QRS_NEXT_CUT()
PTP {E1 29336.867,E2 29336.867}
PTP {X 0,Y 607.919,A -85,B 0,C 180,E1 29336.867,E2 29336.867,E3 0,E4 0,E5 0,E6 0}
QRS_SPEED_INIT()
LIN {X 0,Y 607.919,Z 1319.5,A -85,B 0,C 180,E1 29336.867,E2 29336.867,E3 0,E4 0,E5 0,E6 0} C_VEL
LIN {X 0,Y 607.919,Z 669.088,A -85,B 0,C 180,E1 29336.867,E2 29336.867} C_VEL
LIN {X 0,Y 607.919,Z 661.015,A -85,B 0,C 180,E1 29336.867,E2 29336.867} C_VEL
LIN {X 0,Y 607.916,Z 659.015,A -85,B 0,C 180,E1 29336.679,E2 29336.679} C_VEL
LIN {X 0,Y 607.893,Z 659.005,A -85,B 0,C 180,E1 29333.483,E2 29333.483} C_VEL
LIN {X 0,Y 607.909,Z 659.016,A -85,B 0,C 180,E1 29330.342,E2 29330.342} C_VEL
LIN {X 0,Y 607.894,Z 659.005,A -85,B 0,C 180,E1 29327.171,E2 29327.171} C_VEL
LIN {X 0,Y 607.91,Z 659.015,A -85,B 0,C 180,E1 29323.959,E2 29323.959} C_VEL
LIN {X 0,Y 607.895,Z 659.005,A -85,B 0,C 180,E1 29320.748,E2 29320.748} C_VEL
LIN {X 0,Y 607.917,Z 659.014,A -85,B 0,C 180,E1 29317.564,E2 29317.564} C_VEL
LIN {X 0,Y 607.897,Z 659.005,A -85,B 0,C 180,E1 29314.331,E2 29314.331} C_VEL
LIN {X 0,Y 607.917,Z 659.013,A -85,B 0,C 180,E1 29311.19,E2 29311.19} C_VEL
LIN {X 0,Y 607.905,Z 659.003,A -85,B 0,C 180,E1 29308.021,E2 29308.021} C_VEL
LIN {X 0,Y 607.915,Z 659.014,A -85,B 0,C 180,E1 29304.826,E2 29304.826} C_VEL
LIN {X 0,Y 607.905,Z 659.004,A -85,B 0,C 180,E1 29301.558,E2 29301.558} C_VEL
LIN {X 0,Y 607.904,Z 659.011,A -85,B 0,C 180,E1 29298.305,E2 29298.305} C_VEL
LIN {X 0,Y 607.908,Z 659.004,A -85,B 0,C 180,E1 29295.122,E2 29295.122} C_VEL
LIN {X 0,Y 607.908,Z 659.011,A -85,B 0,C 180,E1 29291.894,E2 29291.894} C_VEL
LIN {X 0,Y 607.911,Z 659.003,A -85,B 0,C 180,E1 29288.681,E2 29288.681} C_VEL
LIN {X 0,Y 607.908,Z 659.008,A -85,B 0,C 180,E1 29285.491,E2 29285.491} C_VEL
LIN {X 0,Y 607.91,Z 658.993,A -85,B 0,C 180,E1 29282.285,E2 29282.285} C_VEL
LIN {X 0,Y 607.909,Z 659.344,A -85,B 0,C 180,E1 29281.725,E2 29281.725} C_VEL
LIN {X 0,Y 607.912,Z 660.667,A -85,B 0,C 180,E1 29281.627,E2 29281.627} C_VEL
LIN {X 0,Y 607.912,Z 878.758,A -85,B 0,C 180,E1 29278.702,E2 29278.702} C_VEL
LIN {X 0,Y 607.912,Z 916.881,A -85,B 0,C 180,E1 29278.166,E2 29278.166} C_VEL
LIN {X 0,Y 607.906,Z 937.091,A -85,B 0,C 180,E1 29277.713,E2 29277.713} C_VEL
LIN {X 0,Y 607.913,Z 958.264,A -85,B 0,C 180,E1 29277.076,E2 29277.076} C_VEL
LIN {X 0,Y 607.913,Z 976.775,A -85,B 0,C 180,E1 29276.364,E2 29276.364} C_VEL
LIN {X 0,Y 607.919,Z 997.894,A -85,B 0,C 180,E1 29275.368,E2 29275.368} C_VEL
LIN {X 0,Y 607.917,Z 1017.228,A -85,B 0,C 180,E1 29274.278,E2 29274.278} C_VEL
LIN {X 0,Y 607.914,Z 1035.659,A -85,B 0,C 180,E1 29273.044,E2 29273.044} C_VEL
LIN {X 0,Y 607.916,Z 1053.23,A -85,B 0,C 180,E1 29271.678,E2 29271.678} C_VEL
LIN {X 0,Y 607.912,Z 1070.203,A -85,B 0,C 180,E1 29270.155,E2 29270.155} C_VEL
LIN {X 0,Y 607.917,Z 1086.083,A -85,B 0,C 180,E1 29268.507,E2 29268.507} C_VEL
LIN {X 0,Y 607.913,Z 1100.76,A -85,B 0,C 180,E1 29266.728,E2 29266.728} C_VEL
LIN {X 0,Y 607.912,Z 1113.249,A -85,B 0,C 180,E1 29264.964,E2 29264.964} C_VEL
LIN {X 0,Y 607.916,Z 1124.49,A -85,B 0,C 180,E1 29263.119,E2 29263.119} C_VEL
LIN {X 0,Y 607.902,Z 1133.845,A -85,B 0,C 180,E1 29261.287,E2 29261.287} C_VEL
LIN {X 0,Y 607.899,Z 1142.297,A -85,B 0,C 180,E1 29259.276,E2 29259.276} C_VEL
LIN {X 0,Y 607.904,Z 1148.818,A -85,B 0,C 180,E1 29257.345,E2 29257.345} C_VEL
LIN {X 0,Y 607.911,Z 1153.711,A -85,B 0,C 180,E1 29255.379,E2 29255.379} C_VEL
LIN {X 0,Y 607.918,Z 1157.29,A -85,B 0,C 180,E1 29253.292,E2 29253.292} C_VEL
LIN {X 0,Y 607.907,Z 1159.182,A -85,B 0,C 180,E1 29251.225,E2 29251.225} C_VEL
LIN {X 0,Y 607.898,Z 1159.339,A -85,B 0,C 180,E1 29249.246,E2 29249.246} C_VEL
LIN {X 0,Y 607.899,Z 1157.836,A -85,B 0,C 180,E1 29247.077,E2 29247.077} C_VEL
LIN {X 0,Y 607.896,Z 1154.903,A -85,B 0,C 180,E1 29245.094,E2 29245.094} C_VEL
LIN {X 0,Y 607.909,Z 1150.265,A -85,B 0,C 180,E1 29243.104,E2 29243.104} C_VEL
LIN {X 0,Y 607.917,Z 1144.051,A -85,B 0,C 180,E1 29241.106,E2 29241.106} C_VEL
LIN {X 0,Y 607.916,Z 1136.441,A -85,B 0,C 180,E1 29239.193,E2 29239.193} C_VEL
LIN {X 0,Y 607.909,Z 1126.947,A -85,B 0,C 180,E1 29237.249,E2 29237.249} C_VEL
LIN {X 0,Y 607.901,Z 1116.406,A -85,B 0,C 180,E1 29235.425,E2 29235.425} C_VEL
LIN {X 0,Y 607.906,Z 1104.361,A -85,B 0,C 180,E1 29233.665,E2 29233.665} C_VEL
LIN {X 0,Y 607.907,Z 1090.255,A -85,B 0,C 180,E1 29231.89,E2 29231.89} C_VEL
LIN {X 0,Y 607.908,Z 1075.163,A -85,B 0,C 180,E1 29230.246,E2 29230.246} C_VEL
LIN {X 0,Y 607.91,Z 1058.641,A -85,B 0,C 180,E1 29228.686,E2 29228.686} C_VEL
LIN {X 0,Y 607.915,Z 1041.052,A -85,B 0,C 180,E1 29227.263,E2 29227.263} C_VEL
LIN {X 0,Y 607.915,Z 1022.644,A -85,B 0,C 180,E1 29225.98,E2 29225.98} C_VEL
LIN {X 0,Y 607.918,Z 1003.587,A -85,B 0,C 180,E1 29224.84,E2 29224.84} C_VEL
LIN {X 0,Y 607.911,Z 984.81,A -85,B 0,C 180,E1 29223.901,E2 29223.901} C_VEL
LIN {X 0,Y 607.918,Z 963.681,A -85,B 0,C 180,E1 29223.03,E2 29223.03} C_VEL
LIN {X 0,Y 607.909,Z 943.544,A -85,B 0,C 180,E1 29222.367,E2 29222.367} C_VEL
LIN {X 0,Y 607.919,Z 923.855,A -85,B 0,C 180,E1 29221.888,E2 29221.888} C_VEL
LIN {X 0,Y 607.905,Z 902.891,A -85,B 0,C 180,E1 29221.526,E2 29221.526} C_VEL
LIN {X 0,Y 607.914,Z 678.859,A -85,B 0,C 180,E1 29218.535,E2 29218.535} C_VEL
LIN {X 0,Y 607.914,Z 659.964,A -85,B 0,C 180,E1 29218.261,E2 29218.261} C_VEL
LIN {X 0,Y 607.909,Z 659.135,A -85,B 0,C 180,E1 29218.133,E2 29218.133} C_VEL
LIN {X 0,Y 607.894,Z 659.003,A -85,B 0,C 180,E1 29215.084,E2 29215.084} C_VEL
LIN {X 0,Y 607.912,Z 659.013,A -85,B 0,C 180,E1 29211.92,E2 29211.92} C_VEL
LIN {X 0,Y 607.898,Z 659.005,A -85,B 0,C 180,E1 29208.735,E2 29208.735} C_VEL
LIN {X 0,Y 607.91,Z 659.013,A -85,B 0,C 180,E1 29205.522,E2 29205.522} C_VEL
LIN {X 0,Y 607.905,Z 659.002,A -85,B 0,C 180,E1 29202.398,E2 29202.398} C_VEL
LIN {X 0,Y 607.909,Z 659.013,A -85,B 0,C 180,E1 29199.167,E2 29199.167} C_VEL
LIN {X 0,Y 607.907,Z 659.003,A -85,B 0,C 180,E1 29195.957,E2 29195.957} C_VEL
LIN {X 0,Y 607.91,Z 659.012,A -85,B 0,C 180,E1 29192.76,E2 29192.76} C_VEL
LIN {X 0,Y 607.912,Z 659.002,A -85,B 0,C 180,E1 29189.537,E2 29189.537} C_VEL
LIN {X 0,Y 607.907,Z 659.01,A -85,B 0,C 180,E1 29186.26,E2 29186.26} C_VEL
LIN {X 0,Y 607.912,Z 659.004,A -85,B 0,C 180,E1 29183.045,E2 29183.045} C_VEL
LIN {X 0,Y 607.908,Z 659.008,A -85,B 0,C 180,E1 29179.805,E2 29179.805} C_VEL
LIN {X 0,Y 607.912,Z 659.005,A -85,B 0,C 180,E1 29176.63,E2 29176.63} C_VEL
LIN {X 0,Y 607.906,Z 659.007,A -85,B 0,C 180,E1 29173.313,E2 29173.313} C_VEL
LIN {X 0,Y 607.912,Z 659.008,A -85,B 0,C 180,E1 29170.041,E2 29170.041} C_VEL
LIN {X 0,Y 607.903,Z 659.005,A -85,B 0,C 180,E1 29166.801,E2 29166.801} C_VEL
LIN {X 0,Y 607.912,Z 659.009,A -85,B 0,C 180,E1 29163.583,E2 29163.583} C_VEL
LIN {X 0,Y 607.906,Z 659.005,A -85,B 0,C 180,E1 29160.377,E2 29160.377} C_VEL
LIN {X 0,Y 607.917,Z 659.011,A -85,B 0,C 180,E1 29157.078,E2 29157.078} C_VEL
LIN {X 0,Y 607.903,Z 659.004,A -85,B 0,C 180,E1 29153.863,E2 29153.863} C_VEL
LIN {X 0,Y 607.919,Z 659.013,A -85,B 0,C 180,E1 29150.629,E2 29150.629} C_VEL
LIN {X 0,Y 607.901,Z 659.003,A -85,B 0,C 180,E1 29147.364,E2 29147.364} C_VEL
LIN {X 0,Y 607.907,Z 659.015,A -85,B 0,C 180,E1 29144.156,E2 29144.156} C_VEL
LIN {X 0,Y 607.901,Z 659.004,A -85,B 0,C 180,E1 29140.895,E2 29140.895} C_VEL
LIN {X 0,Y 607.9,Z 659.013,A -85,B 0,C 180,E1 29137.67,E2 29137.67} C_VEL
LIN {X 0,Y 607.904,Z 659.004,A -85,B 0,C 180,E1 29134.474,E2 29134.474} C_VEL
LIN {X 0,Y 607.904,Z 659.011,A -85,B 0,C 180,E1 29131.239,E2 29131.239} C_VEL
LIN {X 0,Y 607.905,Z 659.005,A -85,B 0,C 180,E1 29128.021,E2 29128.021} C_VEL
LIN {X 0,Y 607.905,Z 659.011,A -85,B 0,C 180,E1 29124.827,E2 29124.827} C_VEL
LIN {X 0,Y 607.908,Z 659.004,A -85,B 0,C 180,E1 29121.677,E2 29121.677} C_VEL
LIN {X 0,Y 607.907,Z 659.006,A -85,B 0,C 180,E1 29118.358,E2 29118.358} C_VEL
LIN {X 0,Y 607.909,Z 659.006,A -85,B 0,C 180,E1 29115.143,E2 29115.143} C_VEL
LIN {X 0,Y 607.908,Z 659.008,A -85,B 0,C 180,E1 29111.894,E2 29111.894} C_VEL
LIN {X 0,Y 607.909,Z 659.002,A -85,B 0,C 180,E1 29108.681,E2 29108.681} C_VEL
LIN {X 0,Y 607.899,Z 659.315,A -85,B 0,C 180,E1 29108.411,E2 29108.411} C_VEL
LIN {X 0,Y 607.916,Z 664.975,A -85,B 0,C 180,E1 29108.018,E2 29108.018} C_VEL
LIN {X 0,Y 607.893,Z 712.988,A -85,B 0,C 180,E1 29105.088,E2 29105.088} C_VEL
LIN {X 0,Y 607.911,Z 759.172,A -85,B 0,C 180,E1 29102.374,E2 29102.374} C_VEL
LIN {X 0,Y 607.916,Z 982.293,A -85,B 0,C 180,E1 29099.362,E2 29099.362} C_VEL
LIN {X 0,Y 607.907,Z 1064.715,A -85,B 0,C 180,E1 29098.246,E2 29098.246} C_VEL
LIN {X 0,Y 607.91,Z 1085.231,A -85,B 0,C 180,E1 29097.805,E2 29097.805} C_VEL
LIN {X 0,Y 607.91,Z 1105.827,A -85,B 0,C 180,E1 29097.208,E2 29097.208} C_VEL
LIN {X 0,Y 607.905,Z 1126.592,A -85,B 0,C 180,E1 29096.417,E2 29096.417} C_VEL
LIN {X 0,Y 607.918,Z 1147.757,A -85,B 0,C 180,E1 29095.421,E2 29095.421} C_VEL
LIN {X 0,Y 607.916,Z 1167.098,A -85,B 0,C 180,E1 29094.332,E2 29094.332} C_VEL
LIN {X 0,Y 607.914,Z 1185.57,A -85,B 0,C 180,E1 29093.095,E2 29093.095} C_VEL
LIN {X 0,Y 607.913,Z 1203.763,A -85,B 0,C 180,E1 29091.678,E2 29091.678} C_VEL
LIN {X 0,Y 607.915,Z 1220.656,A -85,B 0,C 180,E1 29090.155,E2 29090.155} C_VEL
LIN {X 0,Y 607.918,Z 1236.469,A -85,B 0,C 180,E1 29088.507,E2 29088.507} C_VEL
LIN {X 0,Y 607.913,Z 1250.41,A -85,B 0,C 180,E1 29086.817,E2 29086.817} C_VEL
LIN {X 0,Y 607.918,Z 1262.904,A -85,B 0,C 180,E1 29085.062,E2 29085.062} C_VEL
LIN {X 0,Y 607.918,Z 1274.422,A -85,B 0,C 180,E1 29083.176,E2 29083.176} C_VEL
LIN {X 0,Y 607.908,Z 1284.062,A -85,B 0,C 180,E1 29081.287,E2 29081.287} C_VEL
LIN {X 0,Y 607.907,Z 1292.364,A -85,B 0,C 180,E1 29079.302,E2 29079.302} C_VEL
LIN {X 0,Y 607.909,Z 1298.926,A -85,B 0,C 180,E1 29077.351,E2 29077.351} C_VEL
LIN {X 0,Y 607.915,Z 1303.809,A -85,B 0,C 180,E1 29075.379,E2 29075.379} C_VEL
LIN {X 0,Y 607.916,Z 1307.446,A -85,B 0,C 180,E1 29073.206,E2 29073.206} C_VEL
LIN {X 0,Y 607.91,Z 1309.21,A -85,B 0,C 180,E1 29071.225,E2 29071.225} C_VEL
LIN {X 0,Y 607.897,Z 1309.329,A -85,B 0,C 180,E1 29069.246,E2 29069.246} C_VEL
LIN {X 0,Y 607.897,Z 1307.895,A -85,B 0,C 180,E1 29067.172,E2 29067.172} C_VEL
LIN {X 0,Y 607.902,Z 1304.987,A -85,B 0,C 180,E1 29065.188,E2 29065.188} C_VEL
LIN {X 0,Y 607.912,Z 1300.398,A -85,B 0,C 180,E1 29063.199,E2 29063.199} C_VEL
LIN {X 0,Y 607.909,Z 1294.238,A -85,B 0,C 180,E1 29061.202,E2 29061.202} C_VEL
LIN {X 0,Y 607.909,Z 1286.657,A -85,B 0,C 180,E1 29059.289,E2 29059.289} C_VEL
LIN {X 0,Y 607.9,Z 1277.328,A -85,B 0,C 180,E1 29057.364,E2 29057.364} C_VEL
LIN {X 0,Y 607.901,Z 1266.747,A -85,B 0,C 180,E1 29055.523,E2 29055.523} C_VEL
LIN {X 0,Y 607.913,Z 1254.744,A -85,B 0,C 180,E1 29053.764,E2 29053.764} C_VEL
LIN {X 0,Y 607.911,Z 1240.72,A -85,B 0,C 180,E1 29051.989,E2 29051.989} C_VEL
LIN {X 0,Y 607.908,Z 1225.72,A -85,B 0,C 180,E1 29050.346,E2 29050.346} C_VEL
LIN {X 0,Y 607.912,Z 1208.705,A -85,B 0,C 180,E1 29048.737,E2 29048.737} C_VEL
LIN {X 0,Y 607.919,Z 1191.227,A -85,B 0,C 180,E1 29047.322,E2 29047.322} C_VEL
LIN {X 0,Y 607.915,Z 1172.745,A -85,B 0,C 180,E1 29046.031,E2 29046.031} C_VEL
LIN {X 0,Y 607.918,Z 1153.721,A -85,B 0,C 180,E1 29044.892,E2 29044.892} C_VEL
LIN {X 0,Y 607.903,Z 1134.931,A -85,B 0,C 180,E1 29043.951,E2 29043.951} C_VEL
LIN {X 0,Y 607.918,Z 1113.882,A -85,B 0,C 180,E1 29043.082,E2 29043.082} C_VEL
LIN {X 0,Y 607.913,Z 1094.381,A -85,B 0,C 180,E1 29042.438,E2 29042.438} C_VEL
LIN {X 0,Y 607.909,Z 1074.262,A -85,B 0,C 180,E1 29041.941,E2 29041.941} C_VEL
LIN {X 0,Y 607.908,Z 1053.544,A -85,B 0,C 180,E1 29041.58,E2 29041.58} C_VEL
LIN {X 0,Y 607.906,Z 830.992,A -85,B 0,C 180,E1 29038.608,E2 29038.608} C_VEL
LIN {X 0,Y 607.913,Z 758.682,A -85,B 0,C 180,E1 29037.605,E2 29037.605} C_VEL
LIN {X 0,Y 607.904,Z 708.184,A -85,B 0,C 180,E1 29034.624,E2 29034.624} C_VEL
LIN {X 0,Y 607.91,Z 661.098,A -85,B 0,C 180,E1 29031.74,E2 29031.74} C_VEL
LIN {X 0,Y 607.896,Z 659.175,A -85,B 0,C 180,E1 29031.559,E2 29031.559} C_VEL
LIN {X 0,Y 607.894,Z 659.006,A -85,B 0,C 180,E1 29028.592,E2 29028.592} C_VEL
LIN {X 0,Y 607.908,Z 659.015,A -85,B 0,C 180,E1 29025.412,E2 29025.412} C_VEL
LIN {X 0,Y 607.898,Z 659.003,A -85,B 0,C 180,E1 29022.258,E2 29022.258} C_VEL
LIN {X 0,Y 607.91,Z 659.015,A -85,B 0,C 180,E1 29019.045,E2 29019.045} C_VEL
LIN {X 0,Y 607.898,Z 659.005,A -85,B 0,C 180,E1 29015.821,E2 29015.821} C_VEL
LIN {X 0,Y 607.904,Z 659.015,A -85,B 0,C 180,E1 29012.638,E2 29012.638} C_VEL
LIN {X 0,Y 607.905,Z 659.003,A -85,B 0,C 180,E1 29009.458,E2 29009.458} C_VEL
LIN {X 0,Y 607.907,Z 659.013,A -85,B 0,C 180,E1 29006.259,E2 29006.259} C_VEL
LIN {X 0,Y 607.908,Z 659.003,A -85,B 0,C 180,E1 29003.045,E2 29003.045} C_VEL
LIN {X 0,Y 607.908,Z 659.011,A -85,B 0,C 180,E1 28999.805,E2 28999.805} C_VEL
LIN {X 0,Y 607.909,Z 659.004,A -85,B 0,C 180,E1 28996.63,E2 28996.63} C_VEL
LIN {X 0,Y 607.906,Z 659.009,A -85,B 0,C 180,E1 28993.313,E2 28993.313} C_VEL
LIN {X 0,Y 607.911,Z 659.004,A -85,B 0,C 180,E1 28990.136,E2 28990.136} C_VEL
LIN {X 0,Y 607.91,Z 659.008,A -85,B 0,C 180,E1 28986.896,E2 28986.896} C_VEL
LIN {X 0,Y 607.909,Z 659.005,A -85,B 0,C 180,E1 28983.678,E2 28983.678} C_VEL
LIN {X 0,Y 607.906,Z 659.007,A -85,B 0,C 180,E1 28980.377,E2 28980.377} C_VEL
LIN {X 0,Y 607.908,Z 659.007,A -85,B 0,C 180,E1 28977.172,E2 28977.172} C_VEL
LIN {X 0,Y 607.916,Z 659.015,A -85,B 0,C 180,E1 28976.679,E2 28976.679} C_VEL
LIN {X 0,Y 606.925,Z 659.131,A -85,B 0,C 180,E1 28975.953,E2 28975.953} C_VEL
LIN {X 0,Y 600.479,Z 659.931,A -85,B 0,C 180,E1 28973.916,E2 28973.916} C_VEL
LIN {X 0,Y 599.956,Z 659.993,A -85,B 0,C 180,E1 28973.386,E2 28973.386} C_VEL
LIN {X 0,Y 599.974,Z 660.002,A -85,B 0,C 180,E1 28970.213,E2 28970.213} C_VEL
LIN {X 0,Y 599.955,Z 659.994,A -85,B 0,C 180,E1 28966.998,E2 28966.998} C_VEL
LIN {X 0,Y 599.975,Z 660.002,A -85,B 0,C 180,E1 28963.841,E2 28963.841} C_VEL
LIN {X 0,Y 599.954,Z 659.994,A -85,B 0,C 180,E1 28960.603,E2 28960.603} C_VEL
LIN {X 0,Y 599.972,Z 660.001,A -85,B 0,C 180,E1 28957.401,E2 28957.401} C_VEL
LIN {X 0,Y 599.956,Z 659.994,A -85,B 0,C 180,E1 28954.216,E2 28954.216} C_VEL
LIN {X 0,Y 599.969,Z 659.997,A -85,B 0,C 180,E1 28951.032,E2 28951.032} C_VEL
LIN {X 0,Y 599.958,Z 659.993,A -85,B 0,C 180,E1 28947.842,E2 28947.842} C_VEL
LIN {X 0,Y 599.965,Z 659.999,A -85,B 0,C 180,E1 28944.67,E2 28944.67} C_VEL
LIN {X 0,Y 599.96,Z 659.993,A -85,B 0,C 180,E1 28941.443,E2 28941.443} C_VEL
LIN {X 0,Y 599.964,Z 659.998,A -85,B 0,C 180,E1 28938.295,E2 28938.295} C_VEL
LIN {X 0,Y 599.965,Z 659.994,A -85,B 0,C 180,E1 28935.04,E2 28935.04} C_VEL
LIN {X 0,Y 599.963,Z 660,A -85,B 0,C 180,E1 28931.805,E2 28931.805} C_VEL
LIN {X 0,Y 599.968,Z 659.993,A -85,B 0,C 180,E1 28928.593,E2 28928.593} C_VEL
LIN {X 0,Y 599.962,Z 659.992,A -85,B 0,C 180,E1 28925.329,E2 28925.329} C_VEL
LIN {X 0,Y 599.998,Z 660.178,A -85,B 0,C 180,E1 28922.212,E2 28922.212} C_VEL
LIN {X 0,Y 600.395,Z 661.75,A -85,B 0,C 180,E1 28922.054,E2 28922.054} C_VEL
LIN {X 0,Y 601.096,Z 663.832,A -85,B 0,C 180,E1 28921.98,E2 28921.98} C_VEL
LIN {X 0,Y 600.881,Z 888.668,A -85,B 0,C 180,E1 28918.937,E2 28918.937} C_VEL
LIN {X 0,Y 600.837,Z 918.92,A -85,B 0,C 180,E1 28918.486,E2 28918.486} C_VEL
LIN {X 0,Y 600.782,Z 939.065,A -85,B 0,C 180,E1 28918.02,E2 28918.02} C_VEL
LIN {X 0,Y 600.703,Z 960.487,A -85,B 0,C 180,E1 28917.347,E2 28917.347} C_VEL
LIN {X 0,Y 600.631,Z 980.597,A -85,B 0,C 180,E1 28916.548,E2 28916.548} C_VEL
LIN {X 0,Y 600.535,Z 999.897,A -85,B 0,C 180,E1 28915.597,E2 28915.597} C_VEL
LIN {X 0,Y 600.426,Z 1019.653,A -85,B 0,C 180,E1 28914.444,E2 28914.444} C_VEL
LIN {X 0,Y 600.339,Z 1038.558,A -85,B 0,C 180,E1 28913.144,E2 28913.144} C_VEL
LIN {X 0,Y 600.25,Z 1056.372,A -85,B 0,C 180,E1 28911.702,E2 28911.702} C_VEL
LIN {X 0,Y 600.16,Z 1073.033,A -85,B 0,C 180,E1 28910.143,E2 28910.143} C_VEL
LIN {X 0,Y 600.086,Z 1088.641,A -85,B 0,C 180,E1 28908.455,E2 28908.455} C_VEL
LIN {X 0,Y 600.033,Z 1102.301,A -85,B 0,C 180,E1 28906.754,E2 28906.754} C_VEL
LIN {X 0,Y 599.98,Z 1115.257,A -85,B 0,C 180,E1 28904.858,E2 28904.858} C_VEL
LIN {X 0,Y 599.957,Z 1126.572,A -85,B 0,C 180,E1 28902.904,E2 28902.904} C_VEL
LIN {X 0,Y 599.94,Z 1136.062,A -85,B 0,C 180,E1 28900.952,E2 28900.952} C_VEL
LIN {X 0,Y 599.922,Z 1143.719,A -85,B 0,C 180,E1 28899.013,E2 28899.013} C_VEL
LIN {X 0,Y 599.902,Z 1150.026,A -85,B 0,C 180,E1 28896.988,E2 28896.988} C_VEL
LIN {X 0,Y 599.896,Z 1154.739,A -85,B 0,C 180,E1 28894.972,E2 28894.972} C_VEL
LIN {X 0,Y 599.9,Z 1157.73,A -85,B 0,C 180,E1 28892.962,E2 28892.962} C_VEL
LIN {X 0,Y 599.903,Z 1159.296,A -85,B 0,C 180,E1 28890.859,E2 28890.859} C_VEL
LIN {X 0,Y 599.916,Z 1159.25,A -85,B 0,C 180,E1 28888.854,E2 28888.854} C_VEL
LIN {X 0,Y 599.912,Z 1157.612,A -85,B 0,C 180,E1 28886.847,E2 28886.847} C_VEL
LIN {X 0,Y 599.908,Z 1154.317,A -85,B 0,C 180,E1 28884.741,E2 28884.741} C_VEL
LIN {X 0,Y 599.901,Z 1149.755,A -85,B 0,C 180,E1 28882.819,E2 28882.819} C_VEL
LIN {X 0,Y 599.915,Z 1143.339,A -85,B 0,C 180,E1 28880.793,E2 28880.793} C_VEL
LIN {X 0,Y 599.938,Z 1135.624,A -85,B 0,C 180,E1 28878.853,E2 28878.853} C_VEL
LIN {X 0,Y 599.962,Z 1126.01,A -85,B 0,C 180,E1 28876.901,E2 28876.901} C_VEL
LIN {X 0,Y 599.993,Z 1114.479,A -85,B 0,C 180,E1 28874.932,E2 28874.932} C_VEL
LIN {X 0,Y 600.034,Z 1102.229,A -85,B 0,C 180,E1 28873.146,E2 28873.146} C_VEL
LIN {X 0,Y 600.089,Z 1087.699,A -85,B 0,C 180,E1 28871.343,E2 28871.343} C_VEL
LIN {X 0,Y 600.157,Z 1072.482,A -85,B 0,C 180,E1 28869.711,E2 28869.711} C_VEL
LIN {X 0,Y 600.246,Z 1055.016,A -85,B 0,C 180,E1 28868.092,E2 28868.092} C_VEL
LIN {X 0,Y 600.344,Z 1037.658,A -85,B 0,C 180,E1 28866.7,E2 28866.7} C_VEL
LIN {X 0,Y 600.427,Z 1018.619,A -85,B 0,C 180,E1 28865.399,E2 28865.399} C_VEL
LIN {X 0,Y 600.538,Z 998.803,A -85,B 0,C 180,E1 28864.255,E2 28864.255} C_VEL
LIN {X 0,Y 600.638,Z 978.944,A -85,B 0,C 180,E1 28863.292,E2 28863.292} C_VEL
LIN {X 0,Y 600.703,Z 959.315,A -85,B 0,C 180,E1 28862.52,E2 28862.52} C_VEL
LIN {X 0,Y 600.789,Z 937.672,A -85,B 0,C 180,E1 28861.854,E2 28861.854} C_VEL
LIN {X 0,Y 600.851,Z 916.654,A -85,B 0,C 180,E1 28861.378,E2 28861.378} C_VEL
LIN {X 0,Y 600.909,Z 866.117,A -85,B 0,C 180,E1 28860.672,E2 28860.672} C_VEL
LIN {X 0,Y 601.019,Z 663.065,A -85,B 0,C 180,E1 28857.914,E2 28857.914} C_VEL
LIN {X 0,Y 600.049,Z 660.475,A -85,B 0,C 180,E1 28857.771,E2 28857.771} C_VEL
LIN {X 0,Y 599.961,Z 659.966,A -85,B 0,C 180,E1 28857.434,E2 28857.434} C_VEL
LIN {X 0,Y 599.973,Z 659.997,A -85,B 0,C 180,E1 28854.202,E2 28854.202} C_VEL
LIN {X 0,Y 599.963,Z 659.992,A -85,B 0,C 180,E1 28850.951,E2 28850.951} C_VEL
LIN {X 0,Y 599.974,Z 660,A -85,B 0,C 180,E1 28847.682,E2 28847.682} C_VEL
LIN {X 0,Y 599.963,Z 659.994,A -85,B 0,C 180,E1 28844.5,E2 28844.5} C_VEL
LIN {X 0,Y 599.97,Z 660.002,A -85,B 0,C 180,E1 28841.273,E2 28841.273} C_VEL
LIN {X 0,Y 599.966,Z 659.992,A -85,B 0,C 180,E1 28838.069,E2 28838.069} C_VEL
LIN {X 0,Y 599.967,Z 660.001,A -85,B 0,C 180,E1 28834.863,E2 28834.863} C_VEL
LIN {X 0,Y 599.968,Z 659.993,A -85,B 0,C 180,E1 28831.618,E2 28831.618} C_VEL
LIN {X 0,Y 599.964,Z 659.998,A -85,B 0,C 180,E1 28828.357,E2 28828.357} C_VEL
LIN {X 0,Y 599.969,Z 659.994,A -85,B 0,C 180,E1 28825.148,E2 28825.148} C_VEL
LIN {X 0,Y 599.967,Z 659.997,A -85,B 0,C 180,E1 28821.92,E2 28821.92} C_VEL
LIN {X 0,Y 599.973,Z 659.994,A -85,B 0,C 180,E1 28818.762,E2 28818.762} C_VEL
LIN {X 0,Y 599.967,Z 659.996,A -85,B 0,C 180,E1 28815.465,E2 28815.465} C_VEL
LIN {X 0,Y 599.974,Z 659.996,A -85,B 0,C 180,E1 28812.219,E2 28812.219} C_VEL
LIN {X 0,Y 599.968,Z 659.995,A -85,B 0,C 180,E1 28809.013,E2 28809.013} C_VEL
LIN {X 0,Y 599.975,Z 659.996,A -85,B 0,C 180,E1 28805.739,E2 28805.739} C_VEL
LIN {X 0,Y 599.964,Z 659.993,A -85,B 0,C 180,E1 28802.484,E2 28802.484} C_VEL
LIN {X 0,Y 599.976,Z 660,A -85,B 0,C 180,E1 28799.236,E2 28799.236} C_VEL
LIN {X 0,Y 599.963,Z 659.993,A -85,B 0,C 180,E1 28795.987,E2 28795.987} C_VEL
LIN {X 0,Y 599.98,Z 660.002,A -85,B 0,C 180,E1 28792.724,E2 28792.724} C_VEL
LIN {X 0,Y 599.961,Z 659.994,A -85,B 0,C 180,E1 28789.491,E2 28789.491} C_VEL
LIN {X 0,Y 599.969,Z 660.003,A -85,B 0,C 180,E1 28786.3,E2 28786.3} C_VEL
LIN {X 0,Y 599.962,Z 659.994,A -85,B 0,C 180,E1 28783.044,E2 28783.044} C_VEL
LIN {X 0,Y 599.964,Z 660.003,A -85,B 0,C 180,E1 28779.82,E2 28779.82} C_VEL
LIN {X 0,Y 599.965,Z 659.993,A -85,B 0,C 180,E1 28776.632,E2 28776.632} C_VEL
LIN {X 0,Y 599.963,Z 660.001,A -85,B 0,C 180,E1 28773.366,E2 28773.366} C_VEL
LIN {X 0,Y 599.961,Z 659.993,A -85,B 0,C 180,E1 28770.113,E2 28770.113} C_VEL
LIN {X 0,Y 599.961,Z 659.997,A -85,B 0,C 180,E1 28766.865,E2 28766.865} C_VEL
LIN {X 0,Y 599.968,Z 659.995,A -85,B 0,C 180,E1 28763.729,E2 28763.729} C_VEL
LIN {X 0,Y 599.965,Z 659.998,A -85,B 0,C 180,E1 28760.461,E2 28760.461} C_VEL
LIN {X 0,Y 599.966,Z 659.99,A -85,B 0,C 180,E1 28757.291,E2 28757.291} C_VEL
LIN {X 0,Y 599.965,Z 659.996,A -85,B 0,C 180,E1 28754.021,E2 28754.021} C_VEL
LIN {X 0,Y 599.968,Z 659.999,A -85,B 0,C 180,E1 28750.787,E2 28750.787} C_VEL
LIN {X 0,Y 599.995,Z 660.207,A -85,B 0,C 180,E1 28748.966,E2 28748.966} C_VEL
LIN {X 0,Y 601.238,Z 663.981,A -85,B 0,C 180,E1 28748.58,E2 28748.58} C_VEL
LIN {X 0,Y 601.045,Z 711.067,A -85,B 0,C 180,E1 28745.665,E2 28745.665} C_VEL
LIN {X 0,Y 600.978,Z 759.541,A -85,B 0,C 180,E1 28742.787,E2 28742.787} C_VEL
LIN {X 0,Y 600.987,Z 924.529,A -85,B 0,C 180,E1 28740.516,E2 28740.516} C_VEL
LIN {X 0,Y 600.85,Z 1064.826,A -85,B 0,C 180,E1 28738.607,E2 28738.607} C_VEL
LIN {X 0,Y 600.792,Z 1085.937,A -85,B 0,C 180,E1 28738.146,E2 28738.146} C_VEL
LIN {X 0,Y 600.714,Z 1106.568,A -85,B 0,C 180,E1 28737.535,E2 28737.535} C_VEL
LIN {X 0,Y 600.637,Z 1126.595,A -85,B 0,C 180,E1 28736.761,E2 28736.761} C_VEL
LIN {X 0,Y 600.539,Z 1147.933,A -85,B 0,C 180,E1 28735.746,E2 28735.746} C_VEL
LIN {X 0,Y 600.445,Z 1167.12,A -85,B 0,C 180,E1 28734.653,E2 28734.653} C_VEL
LIN {X 0,Y 600.354,Z 1185.421,A -85,B 0,C 180,E1 28733.414,E2 28733.414} C_VEL
LIN {X 0,Y 600.25,Z 1203.28,A -85,B 0,C 180,E1 28732.011,E2 28732.011} C_VEL
LIN {X 0,Y 600.166,Z 1220.15,A -85,B 0,C 180,E1 28730.478,E2 28730.478} C_VEL
LIN {X 0,Y 600.102,Z 1235.664,A -85,B 0,C 180,E1 28728.85,E2 28728.85} C_VEL
LIN {X 0,Y 600.043,Z 1249.563,A -85,B 0,C 180,E1 28727.153,E2 28727.153} C_VEL
LIN {X 0,Y 599.989,Z 1262.905,A -85,B 0,C 180,E1 28725.266,E2 28725.266} C_VEL
LIN {X 0,Y 599.955,Z 1274.213,A -85,B 0,C 180,E1 28723.394,E2 28723.394} C_VEL
LIN {X 0,Y 599.934,Z 1283.827,A -85,B 0,C 180,E1 28721.488,E2 28721.488} C_VEL
LIN {X 0,Y 599.922,Z 1292.11,A -85,B 0,C 180,E1 28719.497,E2 28719.497} C_VEL
LIN {X 0,Y 599.919,Z 1298.873,A -85,B 0,C 180,E1 28717.469,E2 28717.469} C_VEL
LIN {X 0,Y 599.919,Z 1303.809,A -85,B 0,C 180,E1 28715.451,E2 28715.451} C_VEL
LIN {X 0,Y 599.918,Z 1307.446,A -85,B 0,C 180,E1 28713.248,E2 28713.248} C_VEL
LIN {X 0,Y 599.908,Z 1309.21,A -85,B 0,C 180,E1 28711.241,E2 28711.241} C_VEL
LIN {X 0,Y 599.898,Z 1309.329,A -85,B 0,C 180,E1 28709.236,E2 28709.236} C_VEL
LIN {X 0,Y 599.898,Z 1307.895,A -85,B 0,C 180,E1 28707.134,E2 28707.134} C_VEL
LIN {X 0,Y 599.903,Z 1304.987,A -85,B 0,C 180,E1 28705.124,E2 28705.124} C_VEL
LIN {X 0,Y 599.914,Z 1300.398,A -85,B 0,C 180,E1 28703.108,E2 28703.108} C_VEL
LIN {X 0,Y 599.925,Z 1294.239,A -85,B 0,C 180,E1 28701.084,E2 28701.084} C_VEL
LIN {X 0,Y 599.932,Z 1286.658,A -85,B 0,C 180,E1 28699.145,E2 28699.145} C_VEL
LIN {X 0,Y 599.951,Z 1277.07,A -85,B 0,C 180,E1 28697.145,E2 28697.145} C_VEL
LIN {X 0,Y 599.976,Z 1266.112,A -85,B 0,C 180,E1 28695.228,E2 28695.228} C_VEL
LIN {X 0,Y 600.018,Z 1253.496,A -85,B 0,C 180,E1 28693.368,E2 28693.368} C_VEL
LIN {X 0,Y 600.083,Z 1239.871,A -85,B 0,C 180,E1 28691.645,E2 28691.645} C_VEL
LIN {X 0,Y 600.155,Z 1224.2,A -85,B 0,C 180,E1 28689.929,E2 28689.929} C_VEL
LIN {X 0,Y 600.242,Z 1208.108,A -85,B 0,C 180,E1 28688.4,E2 28688.4} C_VEL
LIN {X 0,Y 600.313,Z 1190.47,A -85,B 0,C 180,E1 28686.959,E2 28686.959} C_VEL
LIN {X 0,Y 600.418,Z 1171.865,A -85,B 0,C 180,E1 28685.655,E2 28685.655} C_VEL
LIN {X 0,Y 600.528,Z 1152.127,A -85,B 0,C 180,E1 28684.476,E2 28684.476} C_VEL
LIN {X 0,Y 600.591,Z 1132.695,A -85,B 0,C 180,E1 28683.503,E2 28683.503} C_VEL
LIN {X 0,Y 600.703,Z 1112.452,A -85,B 0,C 180,E1 28682.68,E2 28682.68} C_VEL
LIN {X 0,Y 600.788,Z 1091.832,A -85,B 0,C 180,E1 28682.008,E2 28682.008} C_VEL
LIN {X 0,Y 600.831,Z 1071.411,A -85,B 0,C 180,E1 28681.521,E2 28681.521} C_VEL
LIN {X 0,Y 600.885,Z 1044.281,A -85,B 0,C 180,E1 28681.093,E2 28681.093} C_VEL
LIN {X 0,Y 601.075,Z 818.963,A -85,B 0,C 180,E1 28678.044,E2 28678.044} C_VEL
LIN {X 0,Y 600.962,Z 759.434,A -85,B 0,C 180,E1 28677.21,E2 28677.21} C_VEL
LIN {X 0,Y 601.057,Z 709.241,A -85,B 0,C 180,E1 28674.224,E2 28674.224} C_VEL
LIN {X 0,Y 601.23,Z 663.512,A -85,B 0,C 180,E1 28671.39,E2 28671.39} C_VEL
LIN {X 0,Y 600.008,Z 660.272,A -85,B 0,C 180,E1 28671.051,E2 28671.051} C_VEL
LIN {X 0,Y 599.959,Z 660,A -85,B 0,C 180,E1 28669.459,E2 28669.459} C_VEL
LIN {X 0,Y 599.954,Z 659.994,A -85,B 0,C 180,E1 28666.326,E2 28666.326} C_VEL
LIN {X 0,Y 599.963,Z 659.996,A -85,B 0,C 180,E1 28663.231,E2 28663.231} C_VEL
LIN {X 0,Y 599.957,Z 659.995,A -85,B 0,C 180,E1 28660.037,E2 28660.037} C_VEL
LIN {X 0,Y 599.964,Z 660.004,A -85,B 0,C 180,E1 28656.866,E2 28656.866} C_VEL
LIN {X 0,Y 599.962,Z 659.992,A -85,B 0,C 180,E1 28653.707,E2 28653.707} C_VEL
LIN {X 0,Y 599.96,Z 660.001,A -85,B 0,C 180,E1 28650.439,E2 28650.439} C_VEL
LIN {X 0,Y 599.964,Z 659.994,A -85,B 0,C 180,E1 28647.277,E2 28647.277} C_VEL
LIN {X 0,Y 599.964,Z 660.001,A -85,B 0,C 180,E1 28644.044,E2 28644.044} C_VEL
LIN {X 0,Y 599.964,Z 659.994,A -85,B 0,C 180,E1 28640.789,E2 28640.789} C_VEL
LIN {X 0,Y 599.964,Z 659.999,A -85,B 0,C 180,E1 28637.556,E2 28637.556} C_VEL
LIN {X 0,Y 599.967,Z 659.994,A -85,B 0,C 180,E1 28634.377,E2 28634.377} C_VEL
LIN {X 0,Y 599.967,Z 659.998,A -85,B 0,C 180,E1 28631.146,E2 28631.146} C_VEL
LIN {X 0,Y 599.97,Z 659.994,A -85,B 0,C 180,E1 28627.95,E2 28627.95} C_VEL
LIN {X 0,Y 599.967,Z 659.996,A -85,B 0,C 180,E1 28624.684,E2 28624.684} C_VEL
LIN {X 0,Y 599.972,Z 659.994,A -85,B 0,C 180,E1 28621.528,E2 28621.528} C_VEL
LIN {X 0,Y 599.97,Z 659.995,A -85,B 0,C 180,E1 28618.281,E2 28618.281} C_VEL
LIN {X 0,Y 599.974,Z 659.995,A -85,B 0,C 180,E1 28615.124,E2 28615.124} C_VEL
LIN {X 0,Y 599.956,Z 659.993,A -85,B 0,C 180,E1 28613.386,E2 28613.386} C_VEL
LIN {X 0,Y 598.984,Z 660.123,A -85,B 0,C 180,E1 28612.65,E2 28612.65} C_VEL
LIN {X 0,Y 592.568,Z 660.927,A -85,B 0,C 180,E1 28610.586,E2 28610.586} C_VEL
LIN {X 0,Y 592.036,Z 660.987,A -85,B 0,C 180,E1 28610.049,E2 28610.049} C_VEL
LIN {X 0,Y 592.027,Z 660.984,A -85,B 0,C 180,E1 28606.721,E2 28606.721} C_VEL
LIN {X 0,Y 592.035,Z 660.984,A -85,B 0,C 180,E1 28603.416,E2 28603.416} C_VEL
LIN {X 0,Y 592.03,Z 660.986,A -85,B 0,C 180,E1 28600.156,E2 28600.156} C_VEL
LIN {X 0,Y 592.034,Z 660.981,A -85,B 0,C 180,E1 28596.738,E2 28596.738} C_VEL
LIN {X 0,Y 592.034,Z 660.992,A -85,B 0,C 180,E1 28593.413,E2 28593.413} C_VEL
LIN {X 0,Y 592.021,Z 660.976,A -85,B 0,C 180,E1 28590.117,E2 28590.117} C_VEL
LIN {X 0,Y 592.031,Z 660.991,A -85,B 0,C 180,E1 28586.825,E2 28586.825} C_VEL
LIN {X 0,Y 592.023,Z 660.979,A -85,B 0,C 180,E1 28583.644,E2 28583.644} C_VEL
LIN {X 0,Y 592.029,Z 660.991,A -85,B 0,C 180,E1 28580.453,E2 28580.453} C_VEL
LIN {X 0,Y 592.025,Z 660.977,A -85,B 0,C 180,E1 28577.24,E2 28577.24} C_VEL
LIN {X 0,Y 592.024,Z 660.987,A -85,B 0,C 180,E1 28573.956,E2 28573.956} C_VEL
LIN {X 0,Y 592.026,Z 660.985,A -85,B 0,C 180,E1 28570.684,E2 28570.684} C_VEL
LIN {X 0,Y 592.023,Z 660.989,A -85,B 0,C 180,E1 28567.444,E2 28567.444} C_VEL
LIN {X 0,Y 592.027,Z 660.966,A -85,B 0,C 180,E1 28564.22,E2 28564.22} C_VEL
LIN {X 0,Y 592.047,Z 661.168,A -85,B 0,C 180,E1 28562.682,E2 28562.682} C_VEL
LIN {X 0,Y 592.44,Z 662.686,A -85,B 0,C 180,E1 28562.525,E2 28562.525} C_VEL
LIN {X 0,Y 594.306,Z 666.2,A -85,B 0,C 180,E1 28562.358,E2 28562.358} C_VEL
LIN {X 0,Y 593.876,Z 891.07,A -85,B 0,C 180,E1 28559.28,E2 28559.28} C_VEL
LIN {X 0,Y 593.783,Z 919.716,A -85,B 0,C 180,E1 28558.84,E2 28558.84} C_VEL
LIN {X 0,Y 593.678,Z 940.131,A -85,B 0,C 180,E1 28558.358,E2 28558.358} C_VEL
LIN {X 0,Y 593.513,Z 961.315,A -85,B 0,C 180,E1 28557.677,E2 28557.677} C_VEL
LIN {X 0,Y 593.347,Z 981.752,A -85,B 0,C 180,E1 28556.846,E2 28556.846} C_VEL
LIN {X 0,Y 593.166,Z 1000.907,A -85,B 0,C 180,E1 28555.885,E2 28555.885} C_VEL
LIN {X 0,Y 592.946,Z 1020.468,A -85,B 0,C 180,E1 28554.72,E2 28554.72} C_VEL
LIN {X 0,Y 592.775,Z 1038.984,A -85,B 0,C 180,E1 28553.424,E2 28553.424} C_VEL
LIN {X 0,Y 592.589,Z 1056.695,A -85,B 0,C 180,E1 28551.97,E2 28551.97} C_VEL
LIN {X 0,Y 592.409,Z 1073.252,A -85,B 0,C 180,E1 28550.397,E2 28550.397} C_VEL
LIN {X 0,Y 592.26,Z 1089.497,A -85,B 0,C 180,E1 28548.606,E2 28548.606} C_VEL
LIN {X 0,Y 592.155,Z 1103.018,A -85,B 0,C 180,E1 28546.883,E2 28546.883} C_VEL
LIN {X 0,Y 592.062,Z 1115.825,A -85,B 0,C 180,E1 28544.974,E2 28544.974} C_VEL
LIN {X 0,Y 592.004,Z 1126.576,A -85,B 0,C 180,E1 28543.08,E2 28543.08} C_VEL
LIN {X 0,Y 591.962,Z 1136.136,A -85,B 0,C 180,E1 28541.084,E2 28541.084} C_VEL
LIN {X 0,Y 591.928,Z 1143.722,A -85,B 0,C 180,E1 28539.136,E2 28539.136} C_VEL
LIN {X 0,Y 591.902,Z 1150.028,A -85,B 0,C 180,E1 28537.083,E2 28537.083} C_VEL
LIN {X 0,Y 591.899,Z 1154.741,A -85,B 0,C 180,E1 28535.039,E2 28535.039} C_VEL
LIN {X 0,Y 591.902,Z 1157.732,A -85,B 0,C 180,E1 28533.002,E2 28533.002} C_VEL
LIN {X 0,Y 591.904,Z 1159.296,A -85,B 0,C 180,E1 28530.871,E2 28530.871} C_VEL
LIN {X 0,Y 591.915,Z 1159.25,A -85,B 0,C 180,E1 28528.839,E2 28528.839} C_VEL
LIN {X 0,Y 591.914,Z 1157.611,A -85,B 0,C 180,E1 28526.805,E2 28526.805} C_VEL
LIN {X 0,Y 591.912,Z 1154.316,A -85,B 0,C 180,E1 28524.669,E2 28524.669} C_VEL
LIN {X 0,Y 591.909,Z 1149.754,A -85,B 0,C 180,E1 28522.722,E2 28522.722} C_VEL
LIN {X 0,Y 591.923,Z 1143.337,A -85,B 0,C 180,E1 28520.668,E2 28520.668} C_VEL
LIN {X 0,Y 591.96,Z 1135.621,A -85,B 0,C 180,E1 28518.701,E2 28518.701} C_VEL
LIN {X 0,Y 592.005,Z 1126.007,A -85,B 0,C 180,E1 28516.721,E2 28516.721} C_VEL
LIN {X 0,Y 592.074,Z 1114.476,A -85,B 0,C 180,E1 28514.726,E2 28514.726} C_VEL
LIN {X 0,Y 592.175,Z 1101.921,A -85,B 0,C 180,E1 28512.875,E2 28512.875} C_VEL
LIN {X 0,Y 592.273,Z 1087.694,A -85,B 0,C 180,E1 28511.088,E2 28511.088} C_VEL
LIN {X 0,Y 592.409,Z 1072.618,A -85,B 0,C 180,E1 28509.449,E2 28509.449} C_VEL
LIN {X 0,Y 592.589,Z 1055.858,A -85,B 0,C 180,E1 28507.867,E2 28507.867} C_VEL
LIN {X 0,Y 592.786,Z 1038.365,A -85,B 0,C 180,E1 28506.438,E2 28506.438} C_VEL
LIN {X 0,Y 592.955,Z 1019.407,A -85,B 0,C 180,E1 28505.12,E2 28505.12} C_VEL
LIN {X 0,Y 593.174,Z 999.559,A -85,B 0,C 180,E1 28503.953,E2 28503.953} C_VEL
LIN {X 0,Y 593.378,Z 980.202,A -85,B 0,C 180,E1 28502.993,E2 28502.993} C_VEL
LIN {X 0,Y 593.516,Z 959.939,A -85,B 0,C 180,E1 28502.182,E2 28502.182} C_VEL
LIN {X 0,Y 593.691,Z 937.96,A -85,B 0,C 180,E1 28501.495,E2 28501.495} C_VEL
LIN {X 0,Y 593.813,Z 916.798,A -85,B 0,C 180,E1 28501.01,E2 28501.01} C_VEL
LIN {X 0,Y 593.926,Z 867.527,A -85,B 0,C 180,E1 28500.313,E2 28500.313} C_VEL
LIN {X 0,Y 594.26,Z 665.695,A -85,B 0,C 180,E1 28497.543,E2 28497.543} C_VEL
LIN {X 0,Y 592.225,Z 662.019,A -85,B 0,C 180,E1 28497.353,E2 28497.353} C_VEL
LIN {X 0,Y 592.03,Z 661.065,A -85,B 0,C 180,E1 28497.202,E2 28497.202} C_VEL
LIN {X 0,Y 592.034,Z 660.988,A -85,B 0,C 180,E1 28493.995,E2 28493.995} C_VEL
LIN {X 0,Y 592.019,Z 660.982,A -85,B 0,C 180,E1 28490.824,E2 28490.824} C_VEL
LIN {X 0,Y 592.033,Z 660.986,A -85,B 0,C 180,E1 28487.636,E2 28487.636} C_VEL
LIN {X 0,Y 592.02,Z 660.984,A -85,B 0,C 180,E1 28484.408,E2 28484.408} C_VEL
LIN {X 0,Y 592.027,Z 660.99,A -85,B 0,C 180,E1 28481.198,E2 28481.198} C_VEL
LIN {X 0,Y 592.021,Z 660.983,A -85,B 0,C 180,E1 28477.934,E2 28477.934} C_VEL
LIN {X 0,Y 592.025,Z 660.99,A -85,B 0,C 180,E1 28474.809,E2 28474.809} C_VEL
LIN {X 0,Y 592.028,Z 660.982,A -85,B 0,C 180,E1 28471.571,E2 28471.571} C_VEL
LIN {X 0,Y 592.024,Z 660.987,A -85,B 0,C 180,E1 28468.332,E2 28468.332} C_VEL
LIN {X 0,Y 592.029,Z 660.984,A -85,B 0,C 180,E1 28465.082,E2 28465.082} C_VEL
LIN {X 0,Y 592.022,Z 660.985,A -85,B 0,C 180,E1 28461.812,E2 28461.812} C_VEL
LIN {X 0,Y 592.032,Z 660.985,A -85,B 0,C 180,E1 28458.614,E2 28458.614} C_VEL
LIN {X 0,Y 592.022,Z 660.984,A -85,B 0,C 180,E1 28455.351,E2 28455.351} C_VEL
LIN {X 0,Y 592.033,Z 660.987,A -85,B 0,C 180,E1 28452.088,E2 28452.088} C_VEL
LIN {X 0,Y 592.02,Z 660.984,A -85,B 0,C 180,E1 28448.841,E2 28448.841} C_VEL
LIN {X 0,Y 592.036,Z 660.987,A -85,B 0,C 180,E1 28445.621,E2 28445.621} C_VEL
LIN {X 0,Y 592.022,Z 660.981,A -85,B 0,C 180,E1 28442.42,E2 28442.42} C_VEL
LIN {X 0,Y 592.039,Z 660.991,A -85,B 0,C 180,E1 28439.129,E2 28439.129} C_VEL
LIN {X 0,Y 592.021,Z 660.983,A -85,B 0,C 180,E1 28435.933,E2 28435.933} C_VEL
LIN {X 0,Y 592.041,Z 660.99,A -85,B 0,C 180,E1 28432.723,E2 28432.723} C_VEL
LIN {X 0,Y 592.022,Z 660.983,A -85,B 0,C 180,E1 28429.491,E2 28429.491} C_VEL
LIN {X 0,Y 592.025,Z 660.991,A -85,B 0,C 180,E1 28426.224,E2 28426.224} C_VEL
LIN {X 0,Y 592.022,Z 660.983,A -85,B 0,C 180,E1 28423.012,E2 28423.012} C_VEL
LIN {X 0,Y 592.022,Z 660.991,A -85,B 0,C 180,E1 28419.744,E2 28419.744} C_VEL
LIN {X 0,Y 592.02,Z 660.983,A -85,B 0,C 180,E1 28416.511,E2 28416.511} C_VEL
LIN {X 0,Y 592.022,Z 660.99,A -85,B 0,C 180,E1 28413.303,E2 28413.303} C_VEL
LIN {X 0,Y 592.022,Z 660.981,A -85,B 0,C 180,E1 28410.118,E2 28410.118} C_VEL
LIN {X 0,Y 592.025,Z 660.985,A -85,B 0,C 180,E1 28406.894,E2 28406.894} C_VEL
LIN {X 0,Y 592.025,Z 660.985,A -85,B 0,C 180,E1 28403.665,E2 28403.665} C_VEL
LIN {X 0,Y 592.026,Z 660.987,A -85,B 0,C 180,E1 28400.454,E2 28400.454} C_VEL
LIN {X 0,Y 592.024,Z 660.976,A -85,B 0,C 180,E1 28397.24,E2 28397.24} C_VEL
LIN {X 0,Y 592.023,Z 660.984,A -85,B 0,C 180,E1 28393.956,E2 28393.956} C_VEL
LIN {X 0,Y 592.031,Z 660.988,A -85,B 0,C 180,E1 28390.811,E2 28390.811} C_VEL
LIN {X 0,Y 592.049,Z 661.194,A -85,B 0,C 180,E1 28389.526,E2 28389.526} C_VEL
LIN {X 0,Y 593.518,Z 664.777,A -85,B 0,C 180,E1 28389.125,E2 28389.125} C_VEL
LIN {X 0,Y 594.578,Z 667.825,A -85,B 0,C 180,E1 28388.846,E2 28388.846} C_VEL
LIN {X 0,Y 594.192,Z 714.91,A -85,B 0,C 180,E1 28385.903,E2 28385.903} C_VEL
LIN {X 0,Y 593.997,Z 759.648,A -85,B 0,C 180,E1 28383.219,E2 28383.219} C_VEL
LIN {X 0,Y 594.406,Z 764.258,A -85,B 0,C 180,E1 28383.127,E2 28383.127} C_VEL
LIN {X 0,Y 593.961,Z 998.427,A -85,B 0,C 180,E1 28379.901,E2 28379.901} C_VEL
LIN {X 0,Y 593.816,Z 1066.003,A -85,B 0,C 180,E1 28378.959,E2 28378.959} C_VEL
LIN {X 0,Y 593.692,Z 1086.99,A -85,B 0,C 180,E1 28378.485,E2 28378.485} C_VEL
LIN {X 0,Y 593.523,Z 1108.66,A -85,B 0,C 180,E1 28377.82,E2 28377.82} C_VEL
LIN {X 0,Y 593.374,Z 1129.144,A -85,B 0,C 180,E1 28377.007,E2 28377.007} C_VEL
LIN {X 0,Y 593.177,Z 1148.695,A -85,B 0,C 180,E1 28376.049,E2 28376.049} C_VEL
LIN {X 0,Y 592.971,Z 1168.652,A -85,B 0,C 180,E1 28374.884,E2 28374.884} C_VEL
LIN {X 0,Y 592.795,Z 1187.755,A -85,B 0,C 180,E1 28373.561,E2 28373.561} C_VEL
LIN {X 0,Y 592.588,Z 1205.695,A -85,B 0,C 180,E1 28372.102,E2 28372.102} C_VEL
LIN {X 0,Y 592.413,Z 1222.738,A -85,B 0,C 180,E1 28370.494,E2 28370.494} C_VEL
LIN {X 0,Y 592.269,Z 1238.171,A -85,B 0,C 180,E1 28368.81,E2 28368.81} C_VEL
LIN {X 0,Y 592.17,Z 1251.886,A -85,B 0,C 180,E1 28367.085,E2 28367.085} C_VEL
LIN {X 0,Y 592.073,Z 1264.189,A -85,B 0,C 180,E1 28365.274,E2 28365.274} C_VEL
LIN {X 0,Y 592.005,Z 1275.772,A -85,B 0,C 180,E1 28363.279,E2 28363.279} C_VEL
LIN {X 0,Y 591.963,Z 1285.433,A -85,B 0,C 180,E1 28361.299,E2 28361.299} C_VEL
LIN {X 0,Y 591.931,Z 1293.175,A -85,B 0,C 180,E1 28359.332,E2 28359.332} C_VEL
LIN {X 0,Y 591.913,Z 1299.891,A -85,B 0,C 180,E1 28357.181,E2 28357.181} C_VEL
LIN {X 0,Y 591.908,Z 1304.632,A -85,B 0,C 180,E1 28355.136,E2 28355.136} C_VEL
LIN {X 0,Y 591.909,Z 1307.671,A -85,B 0,C 180,E1 28353.099,E2 28353.099} C_VEL
LIN {X 0,Y 591.908,Z 1309.284,A -85,B 0,C 180,E1 28350.968,E2 28350.968} C_VEL
LIN {X 0,Y 591.913,Z 1309.262,A -85,B 0,C 180,E1 28348.935,E2 28348.935} C_VEL
LIN {X 0,Y 591.915,Z 1307.559,A -85,B 0,C 180,E1 28346.805,E2 28346.805} C_VEL
LIN {X 0,Y 591.915,Z 1304.22,A -85,B 0,C 180,E1 28344.669,E2 28344.669} C_VEL
LIN {X 0,Y 591.914,Z 1299.636,A -85,B 0,C 180,E1 28342.722,E2 28342.722} C_VEL
LIN {X 0,Y 591.931,Z 1293.175,A -85,B 0,C 180,E1 28340.668,E2 28340.668} C_VEL
LIN {X 0,Y 591.963,Z 1285.432,A -85,B 0,C 180,E1 28338.701,E2 28338.701} C_VEL
LIN {X 0,Y 592.005,Z 1275.772,A -85,B 0,C 180,E1 28336.721,E2 28336.721} C_VEL
LIN {X 0,Y 592.074,Z 1264.189,A -85,B 0,C 180,E1 28334.726,E2 28334.726} C_VEL
LIN {X 0,Y 592.171,Z 1251.578,A -85,B 0,C 180,E1 28332.875,E2 28332.875} C_VEL
LIN {X 0,Y 592.278,Z 1237.321,A -85,B 0,C 180,E1 28331.088,E2 28331.088} C_VEL
LIN {X 0,Y 592.416,Z 1222.175,A -85,B 0,C 180,E1 28329.449,E2 28329.449} C_VEL
LIN {X 0,Y 592.595,Z 1204.488,A -85,B 0,C 180,E1 28327.794,E2 28327.794} C_VEL
LIN {X 0,Y 592.797,Z 1187.028,A -85,B 0,C 180,E1 28326.386,E2 28326.386} C_VEL
LIN {X 0,Y 592.971,Z 1168.653,A -85,B 0,C 180,E1 28325.116,E2 28325.116} C_VEL
LIN {X 0,Y 593.177,Z 1148.695,A -85,B 0,C 180,E1 28323.951,E2 28323.951} C_VEL
LIN {X 0,Y 593.374,Z 1129.144,A -85,B 0,C 180,E1 28322.993,E2 28322.993} C_VEL
LIN {X 0,Y 593.523,Z 1108.662,A -85,B 0,C 180,E1 28322.18,E2 28322.18} C_VEL
LIN {X 0,Y 593.692,Z 1086.995,A -85,B 0,C 180,E1 28321.515,E2 28321.515} C_VEL
LIN {X 0,Y 593.816,Z 1066.005,A -85,B 0,C 180,E1 28321.041,E2 28321.041} C_VEL
LIN {X 0,Y 593.967,Z 995.932,A -85,B 0,C 180,E1 28320.065,E2 28320.065} C_VEL
LIN {X 0,Y 594.413,Z 762.043,A -85,B 0,C 180,E1 28316.842,E2 28316.842} C_VEL
LIN {X 0,Y 593.895,Z 758.152,A -85,B 0,C 180,E1 28316.714,E2 28316.714} C_VEL
LIN {X 0,Y 594.271,Z 707.223,A -85,B 0,C 180,E1 28313.625,E2 28313.625} C_VEL
LIN {X 0,Y 594.493,Z 667.139,A -85,B 0,C 180,E1 28311.103,E2 28311.103} C_VEL
LIN {X 0,Y 592.061,Z 661.271,A -85,B 0,C 180,E1 28310.492,E2 28310.492} C_VEL
LIN {X 0,Y 592.033,Z 660.989,A -85,B 0,C 180,E1 28309.166,E2 28309.166} C_VEL
LIN {X 0,Y 592.035,Z 660.985,A -85,B 0,C 180,E1 28305.87,E2 28305.87} C_VEL
LIN {X 0,Y 592.033,Z 660.973,A -85,B 0,C 180,E1 28302.496,E2 28302.496} C_VEL
LIN {X 0,Y 592.042,Z 660.992,A -85,B 0,C 180,E1 28299.17,E2 28299.17} C_VEL
LIN {X 0,Y 592.022,Z 660.984,A -85,B 0,C 180,E1 28295.841,E2 28295.841} C_VEL
LIN {X 0,Y 592.024,Z 660.992,A -85,B 0,C 180,E1 28292.571,E2 28292.571} C_VEL
LIN {X 0,Y 592.02,Z 660.98,A -85,B 0,C 180,E1 28289.326,E2 28289.326} C_VEL
LIN {X 0,Y 592.023,Z 660.989,A -85,B 0,C 180,E1 28286.155,E2 28286.155} C_VEL
LIN {X 0,Y 592.025,Z 660.982,A -85,B 0,C 180,E1 28282.962,E2 28282.962} C_VEL
LIN {X 0,Y 592.026,Z 660.985,A -85,B 0,C 180,E1 28279.741,E2 28279.741} C_VEL
LIN {X 0,Y 592.026,Z 660.984,A -85,B 0,C 180,E1 28276.483,E2 28276.483} C_VEL
LIN {X 0,Y 592.026,Z 660.984,A -85,B 0,C 180,E1 28273.278,E2 28273.278} C_VEL
LIN {X 0,Y 592.025,Z 660.985,A -85,B 0,C 180,E1 28270.018,E2 28270.018} C_VEL
LIN {X 0,Y 592.024,Z 660.985,A -85,B 0,C 180,E1 28266.768,E2 28266.768} C_VEL
LIN {X 0,Y 592.024,Z 660.986,A -85,B 0,C 180,E1 28263.535,E2 28263.535} C_VEL
LIN {X 0,Y 592.023,Z 660.985,A -85,B 0,C 180,E1 28260.29,E2 28260.29} C_VEL
LIN {X 0,Y 592.026,Z 660.985,A -85,B 0,C 180,E1 28257.096,E2 28257.096} C_VEL
LIN {X 0,Y 592.027,Z 660.982,A -85,B 0,C 180,E1 28253.892,E2 28253.892} C_VEL
LIN {X 0,Y 592.029,Z 660.988,A -85,B 0,C 180,E1 28250.669,E2 28250.669} C_VEL
LIN {X 0,Y 592.036,Z 660.987,A -85,B 0,C 180,E1 28250.049,E2 28250.049} C_VEL
LIN {X 0,Y 591.042,Z 661.107,A -85,B 0,C 180,E1 28249.304,E2 28249.304} C_VEL
LIN {X 0,Y 584.604,Z 661.908,A -85,B 0,C 180,E1 28247.212,E2 28247.212} C_VEL
LIN {X 0,Y 584.09,Z 661.973,A -85,B 0,C 180,E1 28246.667,E2 28246.667} C_VEL
LIN {X 0,Y 584.096,Z 661.971,A -85,B 0,C 180,E1 28243.287,E2 28243.287} C_VEL
LIN {X 0,Y 584.095,Z 661.977,A -85,B 0,C 180,E1 28239.979,E2 28239.979} C_VEL
LIN {X 0,Y 584.093,Z 661.97,A -85,B 0,C 180,E1 28236.707,E2 28236.707} C_VEL
LIN {X 0,Y 584.096,Z 661.982,A -85,B 0,C 180,E1 28233.353,E2 28233.353} C_VEL
LIN {X 0,Y 584.083,Z 661.963,A -85,B 0,C 180,E1 28230.122,E2 28230.122} C_VEL
LIN {X 0,Y 584.093,Z 661.98,A -85,B 0,C 180,E1 28226.83,E2 28226.83} C_VEL
LIN {X 0,Y 584.081,Z 661.967,A -85,B 0,C 180,E1 28223.558,E2 28223.558} C_VEL
LIN {X 0,Y 584.083,Z 661.979,A -85,B 0,C 180,E1 28220.318,E2 28220.318} C_VEL
LIN {X 0,Y 584.081,Z 661.966,A -85,B 0,C 180,E1 28217.109,E2 28217.109} C_VEL
LIN {X 0,Y 584.081,Z 661.974,A -85,B 0,C 180,E1 28213.888,E2 28213.888} C_VEL
LIN {X 0,Y 584.087,Z 661.974,A -85,B 0,C 180,E1 28210.682,E2 28210.682} C_VEL
LIN {X 0,Y 584.083,Z 661.979,A -85,B 0,C 180,E1 28207.411,E2 28207.411} C_VEL
LIN {X 0,Y 584.086,Z 661.936,A -85,B 0,C 180,E1 28204.157,E2 28204.157} C_VEL
LIN {X 0,Y 584.112,Z 662.147,A -85,B 0,C 180,E1 28203.17,E2 28203.17} C_VEL
LIN {X 0,Y 584.52,Z 663.744,A -85,B 0,C 180,E1 28203.007,E2 28203.007} C_VEL
LIN {X 0,Y 587.539,Z 669.325,A -85,B 0,C 180,E1 28202.733,E2 28202.733} C_VEL
LIN {X 0,Y 586.89,Z 894.257,A -85,B 0,C 180,E1 28199.62,E2 28199.62} C_VEL
LIN {X 0,Y 586.748,Z 921.532,A -85,B 0,C 180,E1 28199.18,E2 28199.18} C_VEL
LIN {X 0,Y 586.582,Z 942.83,A -85,B 0,C 180,E1 28198.659,E2 28198.659} C_VEL
LIN {X 0,Y 586.334,Z 963.79,A -85,B 0,C 180,E1 28197.953,E2 28197.953} C_VEL
LIN {X 0,Y 586.029,Z 985.04,A -85,B 0,C 180,E1 28197.049,E2 28197.049} C_VEL
LIN {X 0,Y 585.784,Z 1004.866,A -85,B 0,C 180,E1 28196.018,E2 28196.018} C_VEL
LIN {X 0,Y 585.454,Z 1024.492,A -85,B 0,C 180,E1 28194.788,E2 28194.788} C_VEL
LIN {X 0,Y 585.136,Z 1043.059,A -85,B 0,C 180,E1 28193.421,E2 28193.421} C_VEL
LIN {X 0,Y 584.89,Z 1060.346,A -85,B 0,C 180,E1 28191.943,E2 28191.943} C_VEL
LIN {X 0,Y 584.643,Z 1077.234,A -85,B 0,C 180,E1 28190.268,E2 28190.268} C_VEL
LIN {X 0,Y 584.423,Z 1092.053,A -85,B 0,C 180,E1 28188.555,E2 28188.555} C_VEL
LIN {X 0,Y 584.236,Z 1105.851,A -85,B 0,C 180,E1 28186.709,E2 28186.709} C_VEL
LIN {X 0,Y 584.121,Z 1117.668,A -85,B 0,C 180,E1 28184.877,E2 28184.877} C_VEL
LIN {X 0,Y 584.042,Z 1128.138,A -85,B 0,C 180,E1 28182.959,E2 28182.959} C_VEL
LIN {X 0,Y 583.977,Z 1137.699,A -85,B 0,C 180,E1 28180.855,E2 28180.855} C_VEL
LIN {X 0,Y 583.946,Z 1145.107,A -85,B 0,C 180,E1 28178.864,E2 28178.864} C_VEL
LIN {X 0,Y 583.915,Z 1150.792,A -85,B 0,C 180,E1 28176.884,E2 28176.884} C_VEL
LIN {X 0,Y 583.9,Z 1155.391,A -85,B 0,C 180,E1 28174.715,E2 28174.715} C_VEL
LIN {X 0,Y 583.894,Z 1158.182,A -85,B 0,C 180,E1 28172.65,E2 28172.65} C_VEL
LIN {X 0,Y 583.895,Z 1159.363,A -85,B 0,C 180,E1 28170.589,E2 28170.589} C_VEL
LIN {X 0,Y 583.9,Z 1159.112,A -85,B 0,C 180,E1 28168.528,E2 28168.528} C_VEL
LIN {X 0,Y 583.909,Z 1157.274,A -85,B 0,C 180,E1 28166.466,E2 28166.466} C_VEL
LIN {X 0,Y 583.92,Z 1153.698,A -85,B 0,C 180,E1 28164.3,E2 28164.3} C_VEL
LIN {X 0,Y 583.925,Z 1148.721,A -85,B 0,C 180,E1 28162.226,E2 28162.226} C_VEL
LIN {X 0,Y 583.949,Z 1142.271,A -85,B 0,C 180,E1 28160.241,E2 28160.241} C_VEL
LIN {X 0,Y 583.997,Z 1133.809,A -85,B 0,C 180,E1 28158.144,E2 28158.144} C_VEL
LIN {X 0,Y 584.059,Z 1124.447,A -85,B 0,C 180,E1 28156.235,E2 28156.235} C_VEL
LIN {X 0,Y 584.155,Z 1113.191,A -85,B 0,C 180,E1 28154.31,E2 28154.31} C_VEL
LIN {X 0,Y 584.324,Z 1099.904,A -85,B 0,C 180,E1 28152.37,E2 28152.37} C_VEL
LIN {X 0,Y 584.51,Z 1085.983,A -85,B 0,C 180,E1 28150.619,E2 28150.619} C_VEL
LIN {X 0,Y 584.738,Z 1069.85,A -85,B 0,C 180,E1 28148.881,E2 28148.881} C_VEL
LIN {X 0,Y 584.972,Z 1053.619,A -85,B 0,C 180,E1 28147.367,E2 28147.367} C_VEL
LIN {X 0,Y 585.277,Z 1035.464,A -85,B 0,C 180,E1 28145.903,E2 28145.903} C_VEL
LIN {X 0,Y 585.606,Z 1016.348,A -85,B 0,C 180,E1 28144.583,E2 28144.583} C_VEL
LIN {X 0,Y 585.871,Z 996.601,A -85,B 0,C 180,E1 28143.441,E2 28143.441} C_VEL
LIN {X 0,Y 586.17,Z 976.372,A -85,B 0,C 180,E1 28142.468,E2 28142.468} C_VEL
LIN {X 0,Y 586.453,Z 955.531,A -85,B 0,C 180,E1 28141.653,E2 28141.653} C_VEL
LIN {X 0,Y 586.637,Z 934.34,A -85,B 0,C 180,E1 28141.024,E2 28141.024} C_VEL
LIN {X 0,Y 586.822,Z 911.947,A -85,B 0,C 180,E1 28140.551,E2 28140.551} C_VEL
LIN {X 0,Y 587.517,Z 677.305,A -85,B 0,C 180,E1 28137.289,E2 28137.289} C_VEL
LIN {X 0,Y 587.321,Z 668.716,A -85,B 0,C 180,E1 28137.155,E2 28137.155} C_VEL
LIN {X 0,Y 584.247,Z 662.834,A -85,B 0,C 180,E1 28136.855,E2 28136.855} C_VEL
LIN {X 0,Y 584.097,Z 661.99,A -85,B 0,C 180,E1 28136.669,E2 28136.669} C_VEL
LIN {X 0,Y 584.093,Z 661.974,A -85,B 0,C 180,E1 28133.238,E2 28133.238} C_VEL
LIN {X 0,Y 584.096,Z 661.98,A -85,B 0,C 180,E1 28129.923,E2 28129.923} C_VEL
LIN {X 0,Y 584.085,Z 661.969,A -85,B 0,C 180,E1 28126.652,E2 28126.652} C_VEL
LIN {X 0,Y 584.089,Z 661.97,A -85,B 0,C 180,E1 28123.349,E2 28123.349} C_VEL
LIN {X 0,Y 584.08,Z 661.974,A -85,B 0,C 180,E1 28120.065,E2 28120.065} C_VEL
LIN {X 0,Y 584.079,Z 661.972,A -85,B 0,C 180,E1 28116.809,E2 28116.809} C_VEL
LIN {X 0,Y 584.082,Z 661.975,A -85,B 0,C 180,E1 28113.568,E2 28113.568} C_VEL
LIN {X 0,Y 584.078,Z 661.967,A -85,B 0,C 180,E1 28110.331,E2 28110.331} C_VEL
LIN {X 0,Y 584.086,Z 661.974,A -85,B 0,C 180,E1 28107.111,E2 28107.111} C_VEL
LIN {X 0,Y 584.081,Z 661.974,A -85,B 0,C 180,E1 28103.922,E2 28103.922} C_VEL
LIN {X 0,Y 584.091,Z 661.973,A -85,B 0,C 180,E1 28100.754,E2 28100.754} C_VEL
LIN {X 0,Y 584.085,Z 661.974,A -85,B 0,C 180,E1 28097.535,E2 28097.535} C_VEL
LIN {X 0,Y 584.094,Z 661.974,A -85,B 0,C 180,E1 28094.271,E2 28094.271} C_VEL
LIN {X 0,Y 584.084,Z 661.972,A -85,B 0,C 180,E1 28091.054,E2 28091.054} C_VEL
LIN {X 0,Y 584.097,Z 661.977,A -85,B 0,C 180,E1 28087.772,E2 28087.772} C_VEL
LIN {X 0,Y 584.081,Z 661.973,A -85,B 0,C 180,E1 28084.517,E2 28084.517} C_VEL
LIN {X 0,Y 584.099,Z 661.978,A -85,B 0,C 180,E1 28081.177,E2 28081.177} C_VEL
LIN {X 0,Y 584.079,Z 661.971,A -85,B 0,C 180,E1 28077.94,E2 28077.94} C_VEL
LIN {X 0,Y 584.09,Z 661.981,A -85,B 0,C 180,E1 28074.696,E2 28074.696} C_VEL
LIN {X 0,Y 584.079,Z 661.971,A -85,B 0,C 180,E1 28071.534,E2 28071.534} C_VEL
LIN {X 0,Y 584.088,Z 661.977,A -85,B 0,C 180,E1 28068.347,E2 28068.347} C_VEL
LIN {X 0,Y 584.082,Z 661.971,A -85,B 0,C 180,E1 28065.121,E2 28065.121} C_VEL
LIN {X 0,Y 584.08,Z 661.975,A -85,B 0,C 180,E1 28061.847,E2 28061.847} C_VEL
LIN {X 0,Y 584.081,Z 661.973,A -85,B 0,C 180,E1 28058.616,E2 28058.616} C_VEL
LIN {X 0,Y 584.081,Z 661.976,A -85,B 0,C 180,E1 28055.419,E2 28055.419} C_VEL
LIN {X 0,Y 584.083,Z 661.973,A -85,B 0,C 180,E1 28052.25,E2 28052.25} C_VEL
LIN {X 0,Y 584.083,Z 661.978,A -85,B 0,C 180,E1 28048.985,E2 28048.985} C_VEL
LIN {X 0,Y 584.083,Z 661.97,A -85,B 0,C 180,E1 28045.771,E2 28045.771} C_VEL
LIN {X 0,Y 584.085,Z 661.974,A -85,B 0,C 180,E1 28042.577,E2 28042.577} C_VEL
LIN {X 0,Y 584.09,Z 661.974,A -85,B 0,C 180,E1 28039.422,E2 28039.422} C_VEL
LIN {X 0,Y 584.084,Z 661.973,A -85,B 0,C 180,E1 28036.109,E2 28036.109} C_VEL
LIN {X 0,Y 584.086,Z 661.972,A -85,B 0,C 180,E1 28032.89,E2 28032.89} C_VEL
LIN {X 0,Y 584.135,Z 662.221,A -85,B 0,C 180,E1 28030.097,E2 28030.097} C_VEL
LIN {X 0,Y 585.257,Z 665.24,A -85,B 0,C 180,E1 28029.756,E2 28029.756} C_VEL
LIN {X 0,Y 587.931,Z 671.164,A -85,B 0,C 180,E1 28029.151,E2 28029.151} C_VEL
LIN {X 0,Y 587.35,Z 718.754,A -85,B 0,C 180,E1 28026.145,E2 28026.145} C_VEL
LIN {X 0,Y 587.054,Z 759.754,A -85,B 0,C 180,E1 28023.662,E2 28023.662} C_VEL
LIN {X 0,Y 587.701,Z 765.098,A -85,B 0,C 180,E1 28023.543,E2 28023.543} C_VEL
LIN {X 0,Y 587.02,Z 999.724,A -85,B 0,C 180,E1 28020.273,E2 28020.273} C_VEL
LIN {X 0,Y 586.807,Z 1066.214,A -85,B 0,C 180,E1 28019.335,E2 28019.335} C_VEL
LIN {X 0,Y 586.618,Z 1087.418,A -85,B 0,C 180,E1 28018.849,E2 28018.849} C_VEL
LIN {X 0,Y 586.365,Z 1109.255,A -85,B 0,C 180,E1 28018.167,E2 28018.167} C_VEL
LIN {X 0,Y 586.132,Z 1130.409,A -85,B 0,C 180,E1 28017.314,E2 28017.314} C_VEL
LIN {X 0,Y 585.821,Z 1150.748,A -85,B 0,C 180,E1 28016.289,E2 28016.289} C_VEL
LIN {X 0,Y 585.483,Z 1171.147,A -85,B 0,C 180,E1 28015.056,E2 28015.056} C_VEL
LIN {X 0,Y 585.215,Z 1189.801,A -85,B 0,C 180,E1 28013.725,E2 28013.725} C_VEL
LIN {X 0,Y 584.932,Z 1207.508,A -85,B 0,C 180,E1 28012.248,E2 28012.248} C_VEL
LIN {X 0,Y 584.673,Z 1223.465,A -85,B 0,C 180,E1 28010.702,E2 28010.702} C_VEL
LIN {X 0,Y 584.447,Z 1239.535,A -85,B 0,C 180,E1 28008.905,E2 28008.905} C_VEL
LIN {X 0,Y 584.285,Z 1253.334,A -85,B 0,C 180,E1 28007.117,E2 28007.117} C_VEL
LIN {X 0,Y 584.154,Z 1265.473,A -85,B 0,C 180,E1 28005.283,E2 28005.283} C_VEL
LIN {X 0,Y 584.049,Z 1276.292,A -85,B 0,C 180,E1 28003.362,E2 28003.362} C_VEL
LIN {X 0,Y 583.986,Z 1285.844,A -85,B 0,C 180,E1 28001.355,E2 28001.355} C_VEL
LIN {X 0,Y 583.943,Z 1293.53,A -85,B 0,C 180,E1 27999.361,E2 27999.361} C_VEL
LIN {X 0,Y 583.917,Z 1300.145,A -85,B 0,C 180,E1 27997.181,E2 27997.181} C_VEL
LIN {X 0,Y 583.907,Z 1304.825,A -85,B 0,C 180,E1 27995.108,E2 27995.108} C_VEL
LIN {X 0,Y 583.906,Z 1307.784,A -85,B 0,C 180,E1 27993.043,E2 27993.043} C_VEL
LIN {X 0,Y 583.903,Z 1309.306,A -85,B 0,C 180,E1 27990.883,E2 27990.883} C_VEL
LIN {X 0,Y 583.913,Z 1309.239,A -85,B 0,C 180,E1 27988.823,E2 27988.823} C_VEL
LIN {X 0,Y 583.917,Z 1307.559,A -85,B 0,C 180,E1 27986.761,E2 27986.761} C_VEL
LIN {X 0,Y 583.92,Z 1304.22,A -85,B 0,C 180,E1 27984.596,E2 27984.596} C_VEL
LIN {X 0,Y 583.921,Z 1299.636,A -85,B 0,C 180,E1 27982.622,E2 27982.622} C_VEL
LIN {X 0,Y 583.946,Z 1292.989,A -85,B 0,C 180,E1 27980.487,E2 27980.487} C_VEL
LIN {X 0,Y 583.99,Z 1284.983,A -85,B 0,C 180,E1 27978.445,E2 27978.445} C_VEL
LIN {X 0,Y 584.051,Z 1275.254,A -85,B 0,C 180,E1 27976.436,E2 27976.436} C_VEL
LIN {X 0,Y 584.154,Z 1264.126,A -85,B 0,C 180,E1 27974.503,E2 27974.503} C_VEL
LIN {X 0,Y 584.308,Z 1251.884,A -85,B 0,C 180,E1 27972.678,E2 27972.678} C_VEL
LIN {X 0,Y 584.482,Z 1237.322,A -85,B 0,C 180,E1 27970.826,E2 27970.826} C_VEL
LIN {X 0,Y 584.691,Z 1222.175,A -85,B 0,C 180,E1 27969.165,E2 27969.165} C_VEL
LIN {X 0,Y 584.961,Z 1204.49,A -85,B 0,C 180,E1 27967.489,E2 27967.489} C_VEL
LIN {X 0,Y 585.264,Z 1187.013,A -85,B 0,C 180,E1 27966.062,E2 27966.062} C_VEL
LIN {X 0,Y 585.543,Z 1168.736,A -85,B 0,C 180,E1 27964.784,E2 27964.784} C_VEL
LIN {X 0,Y 585.838,Z 1148.763,A -85,B 0,C 180,E1 27963.603,E2 27963.603} C_VEL
LIN {X 0,Y 586.144,Z 1129.147,A -85,B 0,C 180,E1 27962.632,E2 27962.632} C_VEL
LIN {X 0,Y 586.372,Z 1108.784,A -85,B 0,C 180,E1 27961.815,E2 27961.815} C_VEL
LIN {X 0,Y 586.62,Z 1086.905,A -85,B 0,C 180,E1 27961.137,E2 27961.137} C_VEL
LIN {X 0,Y 586.808,Z 1065.684,A -85,B 0,C 180,E1 27960.657,E2 27960.657} C_VEL
LIN {X 0,Y 587.074,Z 980.512,A -85,B 0,C 180,E1 27959.463,E2 27959.463} C_VEL
LIN {X 0,Y 587.689,Z 763.281,A -85,B 0,C 180,E1 27956.43,E2 27956.43} C_VEL
LIN {X 0,Y 586.946,Z 758.152,A -85,B 0,C 180,E1 27956.267,E2 27956.267} C_VEL
LIN {X 0,Y 587.508,Z 706.902,A -85,B 0,C 180,E1 27953.118,E2 27953.118} C_VEL
LIN {X 0,Y 587.857,Z 670.799,A -85,B 0,C 180,E1 27950.819,E2 27950.819} C_VEL
LIN {X 0,Y 584.17,Z 662.422,A -85,B 0,C 180,E1 27949.944,E2 27949.944} C_VEL
LIN {X 0,Y 584.084,Z 661.959,A -85,B 0,C 180,E1 27949.551,E2 27949.551} C_VEL
LIN {X 0,Y 584.077,Z 661.972,A -85,B 0,C 180,E1 27946.381,E2 27946.381} C_VEL
LIN {X 0,Y 584.08,Z 661.963,A -85,B 0,C 180,E1 27943.178,E2 27943.178} C_VEL
LIN {X 0,Y 584.081,Z 661.973,A -85,B 0,C 180,E1 27940.065,E2 27940.065} C_VEL
LIN {X 0,Y 584.083,Z 661.982,A -85,B 0,C 180,E1 27936.808,E2 27936.808} C_VEL
LIN {X 0,Y 584.085,Z 661.968,A -85,B 0,C 180,E1 27933.685,E2 27933.685} C_VEL
LIN {X 0,Y 584.082,Z 661.976,A -85,B 0,C 180,E1 27930.444,E2 27930.444} C_VEL
LIN {X 0,Y 584.083,Z 661.973,A -85,B 0,C 180,E1 27927.197,E2 27927.197} C_VEL
LIN {X 0,Y 584.082,Z 661.977,A -85,B 0,C 180,E1 27923.922,E2 27923.922} C_VEL
LIN {X 0,Y 584.085,Z 661.973,A -85,B 0,C 180,E1 27920.753,E2 27920.753} C_VEL
LIN {X 0,Y 584.085,Z 661.977,A -85,B 0,C 180,E1 27917.534,E2 27917.534} C_VEL
LIN {X 0,Y 584.087,Z 661.972,A -85,B 0,C 180,E1 27914.335,E2 27914.335} C_VEL
LIN {X 0,Y 584.085,Z 661.975,A -85,B 0,C 180,E1 27911.053,E2 27911.053} C_VEL
LIN {X 0,Y 584.087,Z 661.973,A -85,B 0,C 180,E1 27907.871,E2 27907.871} C_VEL
LIN {X 0,Y 584.086,Z 661.974,A -85,B 0,C 180,E1 27904.615,E2 27904.615} C_VEL
LIN {X 0,Y 584.085,Z 661.974,A -85,B 0,C 180,E1 27901.373,E2 27901.373} C_VEL
LIN {X 0,Y 584.085,Z 661.971,A -85,B 0,C 180,E1 27898.136,E2 27898.136} C_VEL
LIN {X 0,Y 584.083,Z 661.978,A -85,B 0,C 180,E1 27894.893,E2 27894.893} C_VEL
LIN {X 0,Y 584.083,Z 661.973,A -85,B 0,C 180,E1 27891.633,E2 27891.633} C_VEL
LIN {X 0,Y 584.089,Z 661.977,A -85,B 0,C 180,E1 27888.446,E2 27888.446} C_VEL
LIN {X 0,Y 584.09,Z 661.973,A -85,B 0,C 180,E1 27886.667,E2 27886.667} C_VEL
LIN {X 0,Y 583.132,Z 662.1,A -85,B 0,C 180,E1 27885.912,E2 27885.912} C_VEL
LIN {X 0,Y 576.61,Z 662.91,A -85,B 0,C 180,E1 27883.736,E2 27883.736} C_VEL
LIN {X 0,Y 576.155,Z 662.96,A -85,B 0,C 180,E1 27883.239,E2 27883.239} C_VEL
LIN {X 0,Y 576.158,Z 662.967,A -85,B 0,C 180,E1 27879.903,E2 27879.903} C_VEL
LIN {X 0,Y 576.147,Z 662.96,A -85,B 0,C 180,E1 27876.583,E2 27876.583} C_VEL
LIN {X 0,Y 576.157,Z 662.969,A -85,B 0,C 180,E1 27873.29,E2 27873.29} C_VEL
LIN {X 0,Y 576.139,Z 662.951,A -85,B 0,C 180,E1 27869.993,E2 27869.993} C_VEL
LIN {X 0,Y 576.15,Z 662.968,A -85,B 0,C 180,E1 27866.743,E2 27866.743} C_VEL
LIN {X 0,Y 576.14,Z 662.956,A -85,B 0,C 180,E1 27863.469,E2 27863.469} C_VEL
LIN {X 0,Y 576.142,Z 662.967,A -85,B 0,C 180,E1 27860.244,E2 27860.244} C_VEL
LIN {X 0,Y 576.14,Z 662.954,A -85,B 0,C 180,E1 27856.997,E2 27856.997} C_VEL
LIN {X 0,Y 576.139,Z 662.962,A -85,B 0,C 180,E1 27853.784,E2 27853.784} C_VEL
LIN {X 0,Y 576.147,Z 662.965,A -85,B 0,C 180,E1 27850.526,E2 27850.526} C_VEL
LIN {X 0,Y 576.14,Z 662.968,A -85,B 0,C 180,E1 27847.276,E2 27847.276} C_VEL
LIN {X 0,Y 576.144,Z 662.906,A -85,B 0,C 180,E1 27844.092,E2 27844.092} C_VEL
LIN {X 0,Y 576.209,Z 663.302,A -85,B 0,C 180,E1 27843.639,E2 27843.639} C_VEL
LIN {X 0,Y 576.782,Z 665.176,A -85,B 0,C 180,E1 27843.484,E2 27843.484} C_VEL
LIN {X 0,Y 580.799,Z 672.178,A -85,B 0,C 180,E1 27843.121,E2 27843.121} C_VEL
LIN {X 0,Y 579.926,Z 897.15,A -85,B 0,C 180,E1 27839.972,E2 27839.972} C_VEL
LIN {X 0,Y 579.74,Z 922.215,A -85,B 0,C 180,E1 27839.554,E2 27839.554} C_VEL
LIN {X 0,Y 579.506,Z 943.507,A -85,B 0,C 180,E1 27839.021,E2 27839.021} C_VEL
LIN {X 0,Y 579.189,Z 963.486,A -85,B 0,C 180,E1 27838.341,E2 27838.341} C_VEL
LIN {X 0,Y 578.824,Z 984.034,A -85,B 0,C 180,E1 27837.465,E2 27837.465} C_VEL
LIN {X 0,Y 578.464,Z 1003.918,A -85,B 0,C 180,E1 27836.428,E2 27836.428} C_VEL
LIN {X 0,Y 578.02,Z 1023.184,A -85,B 0,C 180,E1 27835.219,E2 27835.219} C_VEL
LIN {X 0,Y 577.608,Z 1042.573,A -85,B 0,C 180,E1 27833.786,E2 27833.786} C_VEL
LIN {X 0,Y 577.259,Z 1059.911,A -85,B 0,C 180,E1 27832.291,E2 27832.291} C_VEL
LIN {X 0,Y 576.913,Z 1076.808,A -85,B 0,C 180,E1 27830.598,E2 27830.598} C_VEL
LIN {X 0,Y 576.611,Z 1092.06,A -85,B 0,C 180,E1 27828.815,E2 27828.815} C_VEL
LIN {X 0,Y 576.369,Z 1105.857,A -85,B 0,C 180,E1 27826.944,E2 27826.944} C_VEL
LIN {X 0,Y 576.21,Z 1117.674,A -85,B 0,C 180,E1 27825.086,E2 27825.086} C_VEL
LIN {X 0,Y 576.092,Z 1128.143,A -85,B 0,C 180,E1 27823.141,E2 27823.141} C_VEL
LIN {X 0,Y 576.002,Z 1137.703,A -85,B 0,C 180,E1 27821.008,E2 27821.008} C_VEL
LIN {X 0,Y 575.956,Z 1145.182,A -85,B 0,C 180,E1 27818.965,E2 27818.965} C_VEL
LIN {X 0,Y 575.919,Z 1151.048,A -85,B 0,C 180,E1 27816.88,E2 27816.88} C_VEL
LIN {X 0,Y 575.903,Z 1155.551,A -85,B 0,C 180,E1 27814.68,E2 27814.68} C_VEL
LIN {X 0,Y 575.895,Z 1158.295,A -85,B 0,C 180,E1 27812.587,E2 27812.587} C_VEL
LIN {X 0,Y 575.894,Z 1159.385,A -85,B 0,C 180,E1 27810.497,E2 27810.497} C_VEL
LIN {X 0,Y 575.897,Z 1158.978,A -85,B 0,C 180,E1 27808.309,E2 27808.309} C_VEL
LIN {X 0,Y 575.901,Z 1157.048,A -85,B 0,C 180,E1 27806.217,E2 27806.217} C_VEL
LIN {X 0,Y 575.915,Z 1153.491,A -85,B 0,C 180,E1 27804.121,E2 27804.121} C_VEL
LIN {X 0,Y 575.943,Z 1148.417,A -85,B 0,C 180,E1 27802.017,E2 27802.017} C_VEL
LIN {X 0,Y 575.967,Z 1141.914,A -85,B 0,C 180,E1 27800.003,E2 27800.003} C_VEL
LIN {X 0,Y 576.037,Z 1133.345,A -85,B 0,C 180,E1 27797.877,E2 27797.877} C_VEL
LIN {X 0,Y 576.15,Z 1123.379,A -85,B 0,C 180,E1 27795.837,E2 27795.837} C_VEL
LIN {X 0,Y 576.284,Z 1111.905,A -85,B 0,C 180,E1 27793.883,E2 27793.883} C_VEL
LIN {X 0,Y 576.482,Z 1099.124,A -85,B 0,C 180,E1 27792.018,E2 27792.018} C_VEL
LIN {X 0,Y 576.748,Z 1085.06,A -85,B 0,C 180,E1 27790.242,E2 27790.242} C_VEL
LIN {X 0,Y 577.066,Z 1069.054,A -85,B 0,C 180,E1 27788.503,E2 27788.503} C_VEL
LIN {X 0,Y 577.413,Z 1051.98,A -85,B 0,C 180,E1 27786.909,E2 27786.909} C_VEL
LIN {X 0,Y 577.804,Z 1033.277,A -85,B 0,C 180,E1 27785.408,E2 27785.408} C_VEL
LIN {X 0,Y 578.232,Z 1014.38,A -85,B 0,C 180,E1 27784.113,E2 27784.113} C_VEL
LIN {X 0,Y 578.639,Z 994.576,A -85,B 0,C 180,E1 27782.971,E2 27782.971} C_VEL
LIN {X 0,Y 578.992,Z 973.813,A -85,B 0,C 180,E1 27781.985,E2 27781.985} C_VEL
LIN {X 0,Y 579.381,Z 951.886,A -85,B 0,C 180,E1 27781.155,E2 27781.155} C_VEL
LIN {X 0,Y 579.66,Z 931.143,A -85,B 0,C 180,E1 27780.555,E2 27780.555} C_VEL
LIN {X 0,Y 579.853,Z 909.792,A -85,B 0,C 180,E1 27780.127,E2 27780.127} C_VEL
LIN {X 0,Y 580.773,Z 678.908,A -85,B 0,C 180,E1 27776.885,E2 27776.885} C_VEL
LIN {X 0,Y 580.633,Z 671.537,A -85,B 0,C 180,E1 27776.769,E2 27776.769} C_VEL
LIN {X 0,Y 576.387,Z 664.092,A -85,B 0,C 180,E1 27776.373,E2 27776.373} C_VEL
LIN {X 0,Y 576.163,Z 663.013,A -85,B 0,C 180,E1 27776.209,E2 27776.209} C_VEL
LIN {X 0,Y 576.142,Z 662.966,A -85,B 0,C 180,E1 27772.968,E2 27772.968} C_VEL
LIN {X 0,Y 576.154,Z 662.971,A -85,B 0,C 180,E1 27769.781,E2 27769.781} C_VEL
LIN {X 0,Y 576.14,Z 662.958,A -85,B 0,C 180,E1 27766.504,E2 27766.504} C_VEL
LIN {X 0,Y 576.148,Z 662.956,A -85,B 0,C 180,E1 27763.274,E2 27763.274} C_VEL
LIN {X 0,Y 576.142,Z 662.963,A -85,B 0,C 180,E1 27760.066,E2 27760.066} C_VEL
LIN {X 0,Y 576.14,Z 662.959,A -85,B 0,C 180,E1 27756.779,E2 27756.779} C_VEL
LIN {X 0,Y 576.144,Z 662.963,A -85,B 0,C 180,E1 27753.594,E2 27753.594} C_VEL
LIN {X 0,Y 576.14,Z 662.954,A -85,B 0,C 180,E1 27750.332,E2 27750.332} C_VEL
LIN {X 0,Y 576.147,Z 662.963,A -85,B 0,C 180,E1 27747.096,E2 27747.096} C_VEL
LIN {X 0,Y 576.141,Z 662.963,A -85,B 0,C 180,E1 27743.851,E2 27743.851} C_VEL
LIN {X 0,Y 576.152,Z 662.964,A -85,B 0,C 180,E1 27740.627,E2 27740.627} C_VEL
LIN {X 0,Y 576.141,Z 662.962,A -85,B 0,C 180,E1 27737.357,E2 27737.357} C_VEL
LIN {X 0,Y 576.157,Z 662.967,A -85,B 0,C 180,E1 27734.057,E2 27734.057} C_VEL
LIN {X 0,Y 576.139,Z 662.96,A -85,B 0,C 180,E1 27730.803,E2 27730.803} C_VEL
LIN {X 0,Y 576.162,Z 662.968,A -85,B 0,C 180,E1 27727.579,E2 27727.579} C_VEL
LIN {X 0,Y 576.139,Z 662.962,A -85,B 0,C 180,E1 27724.28,E2 27724.28} C_VEL
LIN {X 0,Y 576.146,Z 662.97,A -85,B 0,C 180,E1 27720.995,E2 27720.995} C_VEL
LIN {X 0,Y 576.14,Z 662.96,A -85,B 0,C 180,E1 27717.812,E2 27717.812} C_VEL
LIN {X 0,Y 576.145,Z 662.969,A -85,B 0,C 180,E1 27714.623,E2 27714.623} C_VEL
LIN {X 0,Y 576.138,Z 662.961,A -85,B 0,C 180,E1 27711.417,E2 27711.417} C_VEL
LIN {X 0,Y 576.141,Z 662.962,A -85,B 0,C 180,E1 27708.169,E2 27708.169} C_VEL
LIN {X 0,Y 576.14,Z 662.961,A -85,B 0,C 180,E1 27705.014,E2 27705.014} C_VEL
LIN {X 0,Y 576.14,Z 662.961,A -85,B 0,C 180,E1 27701.798,E2 27701.798} C_VEL
LIN {X 0,Y 576.142,Z 662.962,A -85,B 0,C 180,E1 27698.627,E2 27698.627} C_VEL
LIN {X 0,Y 576.142,Z 662.964,A -85,B 0,C 180,E1 27695.386,E2 27695.386} C_VEL
LIN {X 0,Y 576.142,Z 662.963,A -85,B 0,C 180,E1 27692.171,E2 27692.171} C_VEL
LIN {X 0,Y 576.144,Z 662.967,A -85,B 0,C 180,E1 27688.975,E2 27688.975} C_VEL
LIN {X 0,Y 576.145,Z 662.958,A -85,B 0,C 180,E1 27685.787,E2 27685.787} C_VEL
LIN {X 0,Y 576.148,Z 662.963,A -85,B 0,C 180,E1 27682.599,E2 27682.599} C_VEL
LIN {X 0,Y 576.15,Z 662.963,A -85,B 0,C 180,E1 27679.4,E2 27679.4} C_VEL
LIN {X 0,Y 576.143,Z 662.958,A -85,B 0,C 180,E1 27676.07,E2 27676.07} C_VEL
LIN {X 0,Y 576.146,Z 662.958,A -85,B 0,C 180,E1 27672.864,E2 27672.864} C_VEL
LIN {X 0,Y 576.184,Z 663.235,A -85,B 0,C 180,E1 27670.695,E2 27670.695} C_VEL
LIN {X 0,Y 577.292,Z 666.173,A -85,B 0,C 180,E1 27670.353,E2 27670.353} C_VEL
LIN {X 0,Y 581.295,Z 674.867,A -85,B 0,C 180,E1 27669.439,E2 27669.439} C_VEL
LIN {X 0,Y 580.532,Z 721.637,A -85,B 0,C 180,E1 27666.454,E2 27666.454} C_VEL
LIN {X 0,Y 580.128,Z 759.721,A -85,B 0,C 180,E1 27664.119,E2 27664.119} C_VEL
LIN {X 0,Y 581.025,Z 766.292,A -85,B 0,C 180,E1 27663.963,E2 27663.963} C_VEL
LIN {X 0,Y 580.104,Z 1001.123,A -85,B 0,C 180,E1 27660.653,E2 27660.653} C_VEL
LIN {X 0,Y 579.825,Z 1066.214,A -85,B 0,C 180,E1 27659.723,E2 27659.723} C_VEL
LIN {X 0,Y 579.569,Z 1087.548,A -85,B 0,C 180,E1 27659.23,E2 27659.23} C_VEL
LIN {X 0,Y 579.256,Z 1108.778,A -85,B 0,C 180,E1 27658.562,E2 27658.562} C_VEL
LIN {X 0,Y 578.938,Z 1129.15,A -85,B 0,C 180,E1 27657.738,E2 27657.738} C_VEL
LIN {X 0,Y 578.527,Z 1148.763,A -85,B 0,C 180,E1 27656.757,E2 27656.757} C_VEL
LIN {X 0,Y 578.138,Z 1168.731,A -85,B 0,C 180,E1 27655.562,E2 27655.562} C_VEL
LIN {X 0,Y 577.737,Z 1187.812,A -85,B 0,C 180,E1 27654.21,E2 27654.21} C_VEL
LIN {X 0,Y 577.326,Z 1205.698,A -85,B 0,C 180,E1 27652.718,E2 27652.718} C_VEL
LIN {X 0,Y 576.973,Z 1222.819,A -85,B 0,C 180,E1 27651.059,E2 27651.059} C_VEL
LIN {X 0,Y 576.677,Z 1238.173,A -85,B 0,C 180,E1 27649.339,E2 27649.339} C_VEL
LIN {X 0,Y 576.443,Z 1252.628,A -85,B 0,C 180,E1 27647.461,E2 27647.461} C_VEL
LIN {X 0,Y 576.237,Z 1264.833,A -85,B 0,C 180,E1 27645.601,E2 27645.601} C_VEL
LIN {X 0,Y 576.096,Z 1276.293,A -85,B 0,C 180,E1 27643.55,E2 27643.55} C_VEL
LIN {X 0,Y 576.013,Z 1285.845,A -85,B 0,C 180,E1 27641.514,E2 27641.514} C_VEL
LIN {X 0,Y 575.957,Z 1293.531,A -85,B 0,C 180,E1 27639.492,E2 27639.492} C_VEL
LIN {X 0,Y 575.923,Z 1300.145,A -85,B 0,C 180,E1 27637.281,E2 27637.281} C_VEL
LIN {X 0,Y 575.911,Z 1304.825,A -85,B 0,C 180,E1 27635.179,E2 27635.179} C_VEL
LIN {X 0,Y 575.908,Z 1307.784,A -85,B 0,C 180,E1 27633.085,E2 27633.085} C_VEL
LIN {X 0,Y 575.904,Z 1309.306,A -85,B 0,C 180,E1 27630.895,E2 27630.895} C_VEL
LIN {X 0,Y 575.911,Z 1309.239,A -85,B 0,C 180,E1 27628.806,E2 27628.806} C_VEL
LIN {X 0,Y 575.917,Z 1307.559,A -85,B 0,C 180,E1 27626.716,E2 27626.716} C_VEL
LIN {X 0,Y 575.922,Z 1304.221,A -85,B 0,C 180,E1 27624.521,E2 27624.521} C_VEL
LIN {X 0,Y 575.932,Z 1299.636,A -85,B 0,C 180,E1 27622.519,E2 27622.519} C_VEL
LIN {X 0,Y 575.96,Z 1293.176,A -85,B 0,C 180,E1 27620.407,E2 27620.407} C_VEL
LIN {X 0,Y 576.019,Z 1285.432,A -85,B 0,C 180,E1 27618.384,E2 27618.384} C_VEL
LIN {X 0,Y 576.101,Z 1275.774,A -85,B 0,C 180,E1 27616.348,E2 27616.348} C_VEL
LIN {X 0,Y 576.243,Z 1264.192,A -85,B 0,C 180,E1 27614.296,E2 27614.296} C_VEL
LIN {X 0,Y 576.453,Z 1251.883,A -85,B 0,C 180,E1 27612.435,E2 27612.435} C_VEL
LIN {X 0,Y 576.7,Z 1237.323,A -85,B 0,C 180,E1 27610.557,E2 27610.557} C_VEL
LIN {X 0,Y 576.989,Z 1222.174,A -85,B 0,C 180,E1 27608.873,E2 27608.873} C_VEL
LIN {X 0,Y 577.348,Z 1204.491,A -85,B 0,C 180,E1 27607.175,E2 27607.175} C_VEL
LIN {X 0,Y 577.745,Z 1186.988,A -85,B 0,C 180,E1 27605.728,E2 27605.728} C_VEL
LIN {X 0,Y 578.138,Z 1168.732,A -85,B 0,C 180,E1 27604.438,E2 27604.438} C_VEL
LIN {X 0,Y 578.527,Z 1148.765,A -85,B 0,C 180,E1 27603.243,E2 27603.243} C_VEL
LIN {X 0,Y 578.938,Z 1129.151,A -85,B 0,C 180,E1 27602.262,E2 27602.262} C_VEL
LIN {X 0,Y 579.256,Z 1108.781,A -85,B 0,C 180,E1 27601.438,E2 27601.438} C_VEL
LIN {X 0,Y 579.574,Z 1086.777,A -85,B 0,C 180,E1 27600.749,E2 27600.749} C_VEL
LIN {X 0,Y 579.828,Z 1065.47,A -85,B 0,C 180,E1 27600.265,E2 27600.265} C_VEL
LIN {X 0,Y 580.258,Z 960.918,A -85,B 0,C 180,E1 27598.787,E2 27598.787} C_VEL
LIN {X 0,Y 580.951,Z 764.39,A -85,B 0,C 180,E1 27596.004,E2 27596.004} C_VEL
LIN {X 0,Y 580.026,Z 758.61,A -85,B 0,C 180,E1 27595.835,E2 27595.835} C_VEL
LIN {X 0,Y 580.776,Z 707.319,A -85,B 0,C 180,E1 27592.645,E2 27592.645} C_VEL
LIN {X 0,Y 581.231,Z 674.474,A -85,B 0,C 180,E1 27590.53,E2 27590.53} C_VEL
LIN {X 0,Y 576.228,Z 663.491,A -85,B 0,C 180,E1 27589.354,E2 27589.354} C_VEL
LIN {X 0,Y 576.158,Z 662.956,A -85,B 0,C 180,E1 27589.008,E2 27589.008} C_VEL
LIN {X 0,Y 576.163,Z 662.966,A -85,B 0,C 180,E1 27585.626,E2 27585.626} C_VEL
LIN {X 0,Y 576.146,Z 662.945,A -85,B 0,C 180,E1 27582.325,E2 27582.325} C_VEL
LIN {X 0,Y 576.154,Z 662.969,A -85,B 0,C 180,E1 27579.046,E2 27579.046} C_VEL
LIN {X 0,Y 576.143,Z 662.963,A -85,B 0,C 180,E1 27575.792,E2 27575.792} C_VEL
LIN {X 0,Y 576.144,Z 662.969,A -85,B 0,C 180,E1 27572.5,E2 27572.5} C_VEL
LIN {X 0,Y 576.142,Z 662.956,A -85,B 0,C 180,E1 27569.3,E2 27569.3} C_VEL
LIN {X 0,Y 576.141,Z 662.964,A -85,B 0,C 180,E1 27566.044,E2 27566.044} C_VEL
LIN {X 0,Y 576.14,Z 662.963,A -85,B 0,C 180,E1 27562.768,E2 27562.768} C_VEL
LIN {X 0,Y 576.141,Z 662.959,A -85,B 0,C 180,E1 27559.556,E2 27559.556} C_VEL
LIN {X 0,Y 576.142,Z 662.964,A -85,B 0,C 180,E1 27556.328,E2 27556.328} C_VEL
LIN {X 0,Y 576.143,Z 662.958,A -85,B 0,C 180,E1 27553.14,E2 27553.14} C_VEL
LIN {X 0,Y 576.143,Z 662.965,A -85,B 0,C 180,E1 27549.893,E2 27549.893} C_VEL
LIN {X 0,Y 576.143,Z 662.963,A -85,B 0,C 180,E1 27546.677,E2 27546.677} C_VEL
LIN {X 0,Y 576.144,Z 662.965,A -85,B 0,C 180,E1 27543.482,E2 27543.482} C_VEL
LIN {X 0,Y 576.142,Z 662.963,A -85,B 0,C 180,E1 27540.199,E2 27540.199} C_VEL
LIN {X 0,Y 576.146,Z 662.963,A -85,B 0,C 180,E1 27537.015,E2 27537.015} C_VEL
LIN {X 0,Y 576.142,Z 662.958,A -85,B 0,C 180,E1 27533.723,E2 27533.723} C_VEL
LIN {X 0,Y 576.15,Z 662.969,A -85,B 0,C 180,E1 27530.51,E2 27530.51} C_VEL
LIN {X 0,Y 576.142,Z 662.961,A -85,B 0,C 180,E1 27527.235,E2 27527.235} C_VEL
LIN {X 0,Y 576.153,Z 662.967,A -85,B 0,C 180,E1 27523.982,E2 27523.982} C_VEL
LIN {X 0,Y 576.155,Z 662.96,A -85,B 0,C 180,E1 27523.239,E2 27523.239} C_VEL
LIN {X 0,Y 575.146,Z 663.087,A -85,B 0,C 180,E1 27522.473,E2 27522.473} C_VEL
LIN {X 0,Y 568.74,Z 663.891,A -85,B 0,C 180,E1 27520.323,E2 27520.323} C_VEL
LIN {X 0,Y 568.221,Z 663.954,A -85,B 0,C 180,E1 27519.763,E2 27519.763} C_VEL
LIN {X 0,Y 568.203,Z 663.949,A -85,B 0,C 180,E1 27516.456,E2 27516.456} C_VEL
LIN {X 0,Y 568.215,Z 663.955,A -85,B 0,C 180,E1 27513.14,E2 27513.14} C_VEL
LIN {X 0,Y 568.199,Z 663.938,A -85,B 0,C 180,E1 27509.9,E2 27509.9} C_VEL
LIN {X 0,Y 568.21,Z 663.957,A -85,B 0,C 180,E1 27506.7,E2 27506.7} C_VEL
LIN {X 0,Y 568.203,Z 663.943,A -85,B 0,C 180,E1 27503.503,E2 27503.503} C_VEL
LIN {X 0,Y 568.204,Z 663.956,A -85,B 0,C 180,E1 27500.26,E2 27500.26} C_VEL
LIN {X 0,Y 568.202,Z 663.941,A -85,B 0,C 180,E1 27497.055,E2 27497.055} C_VEL
LIN {X 0,Y 568.202,Z 663.95,A -85,B 0,C 180,E1 27493.824,E2 27493.824} C_VEL
LIN {X 0,Y 568.209,Z 663.955,A -85,B 0,C 180,E1 27490.52,E2 27490.52} C_VEL
LIN {X 0,Y 568.202,Z 663.958,A -85,B 0,C 180,E1 27487.251,E2 27487.251} C_VEL
LIN {X 0,Y 568.241,Z 664.143,A -85,B 0,C 180,E1 27484.19,E2 27484.19} C_VEL
LIN {X 0,Y 568.658,Z 665.729,A -85,B 0,C 180,E1 27484.023,E2 27484.023} C_VEL
LIN {X 0,Y 574.086,Z 675.255,A -85,B 0,C 180,E1 27483.514,E2 27483.514} C_VEL
LIN {X 0,Y 572.982,Z 900.381,A -85,B 0,C 180,E1 27480.328,E2 27480.328} C_VEL
LIN {X 0,Y 572.756,Z 923.221,A -85,B 0,C 180,E1 27479.929,E2 27479.929} C_VEL
LIN {X 0,Y 572.43,Z 944.959,A -85,B 0,C 180,E1 27479.368,E2 27479.368} C_VEL
LIN {X 0,Y 572.053,Z 965.049,A -85,B 0,C 180,E1 27478.667,E2 27478.667} C_VEL
LIN {X 0,Y 571.548,Z 986.416,A -85,B 0,C 180,E1 27477.725,E2 27477.725} C_VEL
LIN {X 0,Y 571.075,Z 1006.684,A -85,B 0,C 180,E1 27476.628,E2 27476.628} C_VEL
LIN {X 0,Y 570.549,Z 1026.123,A -85,B 0,C 180,E1 27475.37,E2 27475.37} C_VEL
LIN {X 0,Y 570.025,Z 1044.598,A -85,B 0,C 180,E1 27473.955,E2 27473.955} C_VEL
LIN {X 0,Y 569.54,Z 1063.024,A -85,B 0,C 180,E1 27472.305,E2 27472.305} C_VEL
LIN {X 0,Y 569.142,Z 1078.71,A -85,B 0,C 180,E1 27470.677,E2 27470.677} C_VEL
LIN {X 0,Y 568.782,Z 1093.753,A -85,B 0,C 180,E1 27468.871,E2 27468.871} C_VEL
LIN {X 0,Y 568.478,Z 1107.277,A -85,B 0,C 180,E1 27466.975,E2 27466.975} C_VEL
LIN {X 0,Y 568.257,Z 1119.42,A -85,B 0,C 180,E1 27464.989,E2 27464.989} C_VEL
LIN {X 0,Y 568.125,Z 1129.689,A -85,B 0,C 180,E1 27463.018,E2 27463.018} C_VEL
LIN {X 0,Y 568.02,Z 1138.521,A -85,B 0,C 180,E1 27460.959,E2 27460.959} C_VEL
LIN {X 0,Y 567.956,Z 1146.327,A -85,B 0,C 180,E1 27458.708,E2 27458.708} C_VEL
LIN {X 0,Y 567.935,Z 1152.061,A -85,B 0,C 180,E1 27456.571,E2 27456.571} C_VEL
LIN {X 0,Y 567.917,Z 1156.028,A -85,B 0,C 180,E1 27454.443,E2 27454.443} C_VEL
LIN {X 0,Y 567.911,Z 1158.584,A -85,B 0,C 180,E1 27452.22,E2 27452.22} C_VEL
LIN {X 0,Y 567.91,Z 1159.474,A -85,B 0,C 180,E1 27450.101,E2 27450.101} C_VEL
LIN {X 0,Y 567.908,Z 1158.778,A -85,B 0,C 180,E1 27447.982,E2 27447.982} C_VEL
LIN {X 0,Y 567.915,Z 1156.485,A -85,B 0,C 180,E1 27445.76,E2 27445.76} C_VEL
LIN {X 0,Y 567.917,Z 1152.873,A -85,B 0,C 180,E1 27443.734,E2 27443.734} C_VEL
LIN {X 0,Y 567.948,Z 1147.201,A -85,B 0,C 180,E1 27441.496,E2 27441.496} C_VEL
LIN {X 0,Y 568.003,Z 1140.49,A -85,B 0,C 180,E1 27439.452,E2 27439.452} C_VEL
LIN {X 0,Y 568.084,Z 1131.955,A -85,B 0,C 180,E1 27437.394,E2 27437.394} C_VEL
LIN {X 0,Y 568.228,Z 1121.072,A -85,B 0,C 180,E1 27435.218,E2 27435.218} C_VEL
LIN {X 0,Y 568.448,Z 1109.281,A -85,B 0,C 180,E1 27433.235,E2 27433.235} C_VEL
LIN {X 0,Y 568.726,Z 1096.013,A -85,B 0,C 180,E1 27431.34,E2 27431.34} C_VEL
LIN {X 0,Y 569.061,Z 1081.339,A -85,B 0,C 180,E1 27429.535,E2 27429.535} C_VEL
LIN {X 0,Y 569.484,Z 1064.71,A -85,B 0,C 180,E1 27427.769,E2 27427.769} C_VEL
LIN {X 0,Y 569.955,Z 1047.637,A -85,B 0,C 180,E1 27426.205,E2 27426.205} C_VEL
LIN {X 0,Y 570.478,Z 1028.903,A -85,B 0,C 180,E1 27424.74,E2 27424.74} C_VEL
LIN {X 0,Y 570.987,Z 1009.471,A -85,B 0,C 180,E1 27423.451,E2 27423.451} C_VEL
LIN {X 0,Y 571.501,Z 988.426,A -85,B 0,C 180,E1 27422.284,E2 27422.284} C_VEL
LIN {X 0,Y 572.025,Z 967.538,A -85,B 0,C 180,E1 27421.338,E2 27421.338} C_VEL
LIN {X 0,Y 572.396,Z 946.248,A -85,B 0,C 180,E1 27420.583,E2 27420.583} C_VEL
LIN {X 0,Y 572.751,Z 924.103,A -85,B 0,C 180,E1 27420,E2 27420} C_VEL
LIN {X 0,Y 572.975,Z 902.125,A -85,B 0,C 180,E1 27419.607,E2 27419.607} C_VEL
LIN {X 0,Y 574.073,Z 677.966,A -85,B 0,C 180,E1 27416.435,E2 27416.435} C_VEL
LIN {X 0,Y 573.941,Z 674.81,A -85,B 0,C 180,E1 27416.379,E2 27416.379} C_VEL
LIN {X 0,Y 569.561,Z 667.444,A -85,B 0,C 180,E1 27415.977,E2 27415.977} C_VEL
LIN {X 0,Y 568.346,Z 664.683,A -85,B 0,C 180,E1 27415.821,E2 27415.821} C_VEL
LIN {X 0,Y 568.215,Z 663.936,A -85,B 0,C 180,E1 27415.61,E2 27415.61} C_VEL
LIN {X 0,Y 568.22,Z 663.951,A -85,B 0,C 180,E1 27412.242,E2 27412.242} C_VEL
LIN {X 0,Y 568.211,Z 663.951,A -85,B 0,C 180,E1 27408.845,E2 27408.845} C_VEL
LIN {X 0,Y 568.218,Z 663.959,A -85,B 0,C 180,E1 27405.548,E2 27405.548} C_VEL
LIN {X 0,Y 568.201,Z 663.937,A -85,B 0,C 180,E1 27402.2,E2 27402.2} C_VEL
LIN {X 0,Y 568.203,Z 663.952,A -85,B 0,C 180,E1 27398.918,E2 27398.918} C_VEL
LIN {X 0,Y 568.201,Z 663.945,A -85,B 0,C 180,E1 27395.615,E2 27395.615} C_VEL
LIN {X 0,Y 568.2,Z 663.95,A -85,B 0,C 180,E1 27392.34,E2 27392.34} C_VEL
LIN {X 0,Y 568.206,Z 663.94,A -85,B 0,C 180,E1 27389.172,E2 27389.172} C_VEL
LIN {X 0,Y 568.201,Z 663.952,A -85,B 0,C 180,E1 27385.95,E2 27385.95} C_VEL
LIN {X 0,Y 568.213,Z 663.954,A -85,B 0,C 180,E1 27382.667,E2 27382.667} C_VEL
LIN {X 0,Y 568.2,Z 663.95,A -85,B 0,C 180,E1 27379.41,E2 27379.41} C_VEL
LIN {X 0,Y 568.217,Z 663.955,A -85,B 0,C 180,E1 27376.109,E2 27376.109} C_VEL
LIN {X 0,Y 568.202,Z 663.95,A -85,B 0,C 180,E1 27372.81,E2 27372.81} C_VEL
LIN {X 0,Y 568.216,Z 663.959,A -85,B 0,C 180,E1 27369.521,E2 27369.521} C_VEL
LIN {X 0,Y 568.204,Z 663.947,A -85,B 0,C 180,E1 27366.264,E2 27366.264} C_VEL
LIN {X 0,Y 568.21,Z 663.951,A -85,B 0,C 180,E1 27362.925,E2 27362.925} C_VEL
LIN {X 0,Y 568.214,Z 663.952,A -85,B 0,C 180,E1 27359.597,E2 27359.597} C_VEL
LIN {X 0,Y 568.216,Z 663.949,A -85,B 0,C 180,E1 27356.166,E2 27356.166} C_VEL
LIN {X 0,Y 568.224,Z 663.954,A -85,B 0,C 180,E1 27352.722,E2 27352.722} C_VEL
LIN {X 0,Y 568.205,Z 663.95,A -85,B 0,C 180,E1 27349.455,E2 27349.455} C_VEL
LIN {X 0,Y 568.206,Z 663.954,A -85,B 0,C 180,E1 27346.154,E2 27346.154} C_VEL
LIN {X 0,Y 568.202,Z 663.951,A -85,B 0,C 180,E1 27342.911,E2 27342.911} C_VEL
LIN {X 0,Y 568.202,Z 663.956,A -85,B 0,C 180,E1 27339.61,E2 27339.61} C_VEL
LIN {X 0,Y 568.202,Z 663.95,A -85,B 0,C 180,E1 27336.456,E2 27336.456} C_VEL
LIN {X 0,Y 568.204,Z 663.956,A -85,B 0,C 180,E1 27333.226,E2 27333.226} C_VEL
LIN {X 0,Y 568.2,Z 663.946,A -85,B 0,C 180,E1 27329.968,E2 27329.968} C_VEL
LIN {X 0,Y 568.201,Z 663.948,A -85,B 0,C 180,E1 27326.7,E2 27326.7} C_VEL
LIN {X 0,Y 568.203,Z 663.956,A -85,B 0,C 180,E1 27323.504,E2 27323.504} C_VEL
LIN {X 0,Y 568.202,Z 663.954,A -85,B 0,C 180,E1 27320.261,E2 27320.261} C_VEL
LIN {X 0,Y 568.199,Z 663.93,A -85,B 0,C 180,E1 27317.055,E2 27317.055} C_VEL
LIN {X 0,Y 568.202,Z 663.95,A -85,B 0,C 180,E1 27313.824,E2 27313.824} C_VEL
LIN {X 0,Y 568.244,Z 664.235,A -85,B 0,C 180,E1 27311.313,E2 27311.313} C_VEL
LIN {X 0,Y 569.799,Z 667.825,A -85,B 0,C 180,E1 27310.882,E2 27310.882} C_VEL
LIN {X 0,Y 574.673,Z 678.569,A -85,B 0,C 180,E1 27309.734,E2 27309.734} C_VEL
LIN {X 0,Y 573.715,Z 725.481,A -85,B 0,C 180,E1 27306.709,E2 27306.709} C_VEL
LIN {X 0,Y 573.238,Z 759.755,A -85,B 0,C 180,E1 27304.586,E2 27304.586} C_VEL
LIN {X 0,Y 574.38,Z 767.677,A -85,B 0,C 180,E1 27304.39,E2 27304.39} C_VEL
LIN {X 0,Y 573.212,Z 1003.108,A -85,B 0,C 180,E1 27301.034,E2 27301.034} C_VEL
LIN {X 0,Y 572.869,Z 1066.413,A -85,B 0,C 180,E1 27300.117,E2 27300.117} C_VEL
LIN {X 0,Y 572.545,Z 1087.808,A -85,B 0,C 180,E1 27299.617,E2 27299.617} C_VEL
LIN {X 0,Y 572.145,Z 1109.592,A -85,B 0,C 180,E1 27298.919,E2 27298.919} C_VEL
LIN {X 0,Y 571.736,Z 1130.41,A -85,B 0,C 180,E1 27298.061,E2 27298.061} C_VEL
LIN {X 0,Y 571.224,Z 1149.76,A -85,B 0,C 180,E1 27297.07,E2 27297.07} C_VEL
LIN {X 0,Y 570.706,Z 1170.158,A -85,B 0,C 180,E1 27295.821,E2 27295.821} C_VEL
LIN {X 0,Y 570.198,Z 1189.127,A -85,B 0,C 180,E1 27294.445,E2 27294.445} C_VEL
LIN {X 0,Y 569.698,Z 1206.907,A -85,B 0,C 180,E1 27292.93,E2 27292.93} C_VEL
LIN {X 0,Y 569.261,Z 1223.534,A -85,B 0,C 180,E1 27291.282,E2 27291.282} C_VEL
LIN {X 0,Y 568.877,Z 1239.024,A -85,B 0,C 180,E1 27289.508,E2 27289.508} C_VEL
LIN {X 0,Y 568.577,Z 1253.279,A -85,B 0,C 180,E1 27287.614,E2 27287.614} C_VEL
LIN {X 0,Y 568.324,Z 1265.471,A -85,B 0,C 180,E1 27285.719,E2 27285.719} C_VEL
LIN {X 0,Y 568.152,Z 1276.366,A -85,B 0,C 180,E1 27283.729,E2 27283.729} C_VEL
LIN {X 0,Y 568.044,Z 1285.846,A -85,B 0,C 180,E1 27281.678,E2 27281.678} C_VEL
LIN {X 0,Y 567.974,Z 1293.531,A -85,B 0,C 180,E1 27279.627,E2 27279.627} C_VEL
LIN {X 0,Y 567.929,Z 1300.145,A -85,B 0,C 180,E1 27277.384,E2 27277.384} C_VEL
LIN {X 0,Y 567.915,Z 1304.825,A -85,B 0,C 180,E1 27275.253,E2 27275.253} C_VEL
LIN {X 0,Y 567.911,Z 1307.784,A -85,B 0,C 180,E1 27273.129,E2 27273.129} C_VEL
LIN {X 0,Y 567.905,Z 1309.306,A -85,B 0,C 180,E1 27270.908,E2 27270.908} C_VEL
LIN {X 0,Y 567.91,Z 1309.239,A -85,B 0,C 180,E1 27268.789,E2 27268.789} C_VEL
LIN {X 0,Y 567.915,Z 1307.486,A -85,B 0,C 180,E1 27266.604,E2 27266.604} C_VEL
LIN {X 0,Y 567.922,Z 1304.015,A -85,B 0,C 180,E1 27264.342,E2 27264.342} C_VEL
LIN {X 0,Y 567.945,Z 1299.128,A -85,B 0,C 180,E1 27262.209,E2 27262.209} C_VEL
LIN {X 0,Y 567.985,Z 1292.466,A -85,B 0,C 180,E1 27260.066,E2 27260.066} C_VEL
LIN {X 0,Y 568.07,Z 1284.064,A -85,B 0,C 180,E1 27257.91,E2 27257.91} C_VEL
LIN {X 0,Y 568.203,Z 1274.164,A -85,B 0,C 180,E1 27255.832,E2 27255.832} C_VEL
LIN {X 0,Y 568.379,Z 1262.767,A -85,B 0,C 180,E1 27253.839,E2 27253.839} C_VEL
LIN {X 0,Y 568.641,Z 1249.568,A -85,B 0,C 180,E1 27251.868,E2 27251.868} C_VEL
LIN {X 0,Y 568.971,Z 1235.589,A -85,B 0,C 180,E1 27250.068,E2 27250.068} C_VEL
LIN {X 0,Y 569.355,Z 1220.148,A -85,B 0,C 180,E1 27248.36,E2 27248.36} C_VEL
LIN {X 0,Y 569.795,Z 1203.285,A -85,B 0,C 180,E1 27246.746,E2 27246.746} C_VEL
LIN {X 0,Y 570.308,Z 1184.24,A -85,B 0,C 180,E1 27245.182,E2 27245.182} C_VEL
LIN {X 0,Y 570.847,Z 1165.432,A -85,B 0,C 180,E1 27243.864,E2 27243.864} C_VEL
LIN {X 0,Y 571.342,Z 1145.771,A -85,B 0,C 180,E1 27242.71,E2 27242.71} C_VEL
LIN {X 0,Y 571.808,Z 1125.335,A -85,B 0,C 180,E1 27241.715,E2 27241.715} C_VEL
LIN {X 0,Y 572.288,Z 1104.338,A -85,B 0,C 180,E1 27240.891,E2 27240.891} C_VEL
LIN {X 0,Y 572.601,Z 1083.267,A -85,B 0,C 180,E1 27240.26,E2 27240.26} C_VEL
LIN {X 0,Y 572.897,Z 1061.146,A -85,B 0,C 180,E1 27239.795,E2 27239.795} C_VEL
LIN {X 0,Y 574.036,Z 833.081,A -85,B 0,C 180,E1 27236.552,E2 27236.552} C_VEL
LIN {X 0,Y 574.198,Z 765.204,A -85,B 0,C 180,E1 27235.561,E2 27235.561} C_VEL
LIN {X 0,Y 573.135,Z 758.687,A -85,B 0,C 180,E1 27235.371,E2 27235.371} C_VEL
LIN {X 0,Y 574.094,Z 707.127,A -85,B 0,C 180,E1 27232.121,E2 27232.121} C_VEL
LIN {X 0,Y 574.673,Z 678.569,A -85,B 0,C 180,E1 27230.266,E2 27230.266} C_VEL
LIN {X 0,Y 568.268,Z 664.374,A -85,B 0,C 180,E1 27228.716,E2 27228.716} C_VEL
LIN {X 0,Y 568.207,Z 663.958,A -85,B 0,C 180,E1 27228.253,E2 27228.253} C_VEL
LIN {X 0,Y 568.213,Z 663.952,A -85,B 0,C 180,E1 27224.879,E2 27224.879} C_VEL
LIN {X 0,Y 568.214,Z 663.936,A -85,B 0,C 180,E1 27221.559,E2 27221.559} C_VEL
LIN {X 0,Y 568.215,Z 663.946,A -85,B 0,C 180,E1 27218.137,E2 27218.137} C_VEL
LIN {X 0,Y 568.21,Z 663.953,A -85,B 0,C 180,E1 27214.741,E2 27214.741} C_VEL
LIN {X 0,Y 568.203,Z 663.952,A -85,B 0,C 180,E1 27211.414,E2 27211.414} C_VEL
LIN {X 0,Y 568.201,Z 663.957,A -85,B 0,C 180,E1 27208.138,E2 27208.138} C_VEL
LIN {X 0,Y 568.201,Z 663.949,A -85,B 0,C 180,E1 27204.87,E2 27204.87} C_VEL
LIN {X 0,Y 568.202,Z 663.954,A -85,B 0,C 180,E1 27201.687,E2 27201.687} C_VEL
LIN {X 0,Y 568.202,Z 663.945,A -85,B 0,C 180,E1 27198.466,E2 27198.466} C_VEL
LIN {X 0,Y 568.203,Z 663.951,A -85,B 0,C 180,E1 27195.2,E2 27195.2} C_VEL
LIN {X 0,Y 568.201,Z 663.947,A -85,B 0,C 180,E1 27191.984,E2 27191.984} C_VEL
LIN {X 0,Y 568.2,Z 663.951,A -85,B 0,C 180,E1 27188.704,E2 27188.704} C_VEL
LIN {X 0,Y 568.203,Z 663.954,A -85,B 0,C 180,E1 27185.554,E2 27185.554} C_VEL
LIN {X 0,Y 568.202,Z 663.95,A -85,B 0,C 180,E1 27182.319,E2 27182.319} C_VEL
LIN {X 0,Y 568.205,Z 663.957,A -85,B 0,C 180,E1 27179.092,E2 27179.092} C_VEL
LIN {X 0,Y 568.203,Z 663.951,A -85,B 0,C 180,E1 27175.863,E2 27175.863} C_VEL
LIN {X 0,Y 568.208,Z 663.953,A -85,B 0,C 180,E1 27172.619,E2 27172.619} C_VEL
LIN {X 0,Y 568.202,Z 663.948,A -85,B 0,C 180,E1 27169.352,E2 27169.352} C_VEL
LIN {X 0,Y 568.218,Z 663.959,A -85,B 0,C 180,E1 27166.05,E2 27166.05} C_VEL
LIN {X 0,Y 568.201,Z 663.95,A -85,B 0,C 180,E1 27162.699,E2 27162.699} C_VEL
LIN {X 0,Y 568.221,Z 663.954,A -85,B 0,C 180,E1 27159.763,E2 27159.763} C_VEL
LIN {X 0,Y 567.238,Z 664.076,A -85,B 0,C 180,E1 27158.986,E2 27158.986} C_VEL
LIN {X 0,Y 560.79,Z 664.875,A -85,B 0,C 180,E1 27156.806,E2 27156.806} C_VEL
LIN {X 0,Y 560.263,Z 664.939,A -85,B 0,C 180,E1 27156.238,E2 27156.238} C_VEL
LIN {X 0,Y 560.273,Z 664.941,A -85,B 0,C 180,E1 27152.93,E2 27152.93} C_VEL
LIN {X 0,Y 560.262,Z 664.926,A -85,B 0,C 180,E1 27149.665,E2 27149.665} C_VEL
LIN {X 0,Y 560.27,Z 664.942,A -85,B 0,C 180,E1 27146.411,E2 27146.411} C_VEL
LIN {X 0,Y 560.267,Z 664.931,A -85,B 0,C 180,E1 27143.081,E2 27143.081} C_VEL
LIN {X 0,Y 560.282,Z 664.938,A -85,B 0,C 180,E1 27139.64,E2 27139.64} C_VEL
LIN {X 0,Y 560.273,Z 664.939,A -85,B 0,C 180,E1 27136.178,E2 27136.178} C_VEL
LIN {X 0,Y 560.269,Z 664.934,A -85,B 0,C 180,E1 27132.822,E2 27132.822} C_VEL
LIN {X 0,Y 560.265,Z 664.939,A -85,B 0,C 180,E1 27129.56,E2 27129.56} C_VEL
LIN {X 0,Y 560.272,Z 664.941,A -85,B 0,C 180,E1 27126.332,E2 27126.332} C_VEL
LIN {X 0,Y 560.299,Z 665.149,A -85,B 0,C 180,E1 27124.728,E2 27124.728} C_VEL
LIN {X 0,Y 560.701,Z 666.66,A -85,B 0,C 180,E1 27124.561,E2 27124.561} C_VEL
LIN {X 0,Y 567.401,Z 678.254,A -85,B 0,C 180,E1 27123.919,E2 27123.919} C_VEL
LIN {X 0,Y 566.064,Z 903.357,A -85,B 0,C 180,E1 27120.696,E2 27120.696} C_VEL
LIN {X 0,Y 565.79,Z 925.037,A -85,B 0,C 180,E1 27120.296,E2 27120.296} C_VEL
LIN {X 0,Y 565.346,Z 947.34,A -85,B 0,C 180,E1 27119.693,E2 27119.693} C_VEL
LIN {X 0,Y 564.918,Z 967.916,A -85,B 0,C 180,E1 27118.951,E2 27118.951} C_VEL
LIN {X 0,Y 564.297,Z 988.549,A -85,B 0,C 180,E1 27118.004,E2 27118.004} C_VEL
LIN {X 0,Y 563.691,Z 1009.175,A -85,B 0,C 180,E1 27116.848,E2 27116.848} C_VEL
LIN {X 0,Y 563.072,Z 1028.428,A -85,B 0,C 180,E1 27115.562,E2 27115.562} C_VEL
LIN {X 0,Y 562.449,Z 1046.561,A -85,B 0,C 180,E1 27114.133,E2 27114.133} C_VEL
LIN {X 0,Y 561.893,Z 1063.765,A -85,B 0,C 180,E1 27112.551,E2 27112.551} C_VEL
LIN {X 0,Y 561.363,Z 1080.588,A -85,B 0,C 180,E1 27110.757,E2 27110.757} C_VEL
LIN {X 0,Y 560.94,Z 1095.364,A -85,B 0,C 180,E1 27108.929,E2 27108.929} C_VEL
LIN {X 0,Y 560.584,Z 1108.685,A -85,B 0,C 180,E1 27107.008,E2 27107.008} C_VEL
LIN {X 0,Y 560.318,Z 1120.578,A -85,B 0,C 180,E1 27104.995,E2 27104.995} C_VEL
LIN {X 0,Y 560.143,Z 1131.095,A -85,B 0,C 180,E1 27102.892,E2 27102.892} C_VEL
LIN {X 0,Y 560.031,Z 1139.741,A -85,B 0,C 180,E1 27100.804,E2 27100.804} C_VEL
LIN {X 0,Y 559.96,Z 1146.936,A -85,B 0,C 180,E1 27098.626,E2 27098.626} C_VEL
LIN {X 0,Y 559.931,Z 1152.485,A -85,B 0,C 180,E1 27096.459,E2 27096.459} C_VEL
LIN {X 0,Y 559.917,Z 1156.188,A -85,B 0,C 180,E1 27094.404,E2 27094.404} C_VEL
LIN {X 0,Y 559.911,Z 1158.652,A -85,B 0,C 180,E1 27092.149,E2 27092.149} C_VEL
LIN {X 0,Y 559.912,Z 1159.496,A -85,B 0,C 180,E1 27090,E2 27090} C_VEL
LIN {X 0,Y 559.914,Z 1158.711,A -85,B 0,C 180,E1 27087.851,E2 27087.851} C_VEL
LIN {X 0,Y 559.918,Z 1156.326,A -85,B 0,C 180,E1 27085.596,E2 27085.596} C_VEL
LIN {X 0,Y 559.93,Z 1152.665,A -85,B 0,C 180,E1 27083.541,E2 27083.541} C_VEL
LIN {X 0,Y 559.96,Z 1147.199,A -85,B 0,C 180,E1 27081.374,E2 27081.374} C_VEL
LIN {X 0,Y 560.031,Z 1140.092,A -85,B 0,C 180,E1 27079.196,E2 27079.196} C_VEL
LIN {X 0,Y 560.138,Z 1131.49,A -85,B 0,C 180,E1 27077.108,E2 27077.108} C_VEL
LIN {X 0,Y 560.31,Z 1121.069,A -85,B 0,C 180,E1 27075.005,E2 27075.005} C_VEL
LIN {X 0,Y 560.573,Z 1109.275,A -85,B 0,C 180,E1 27072.992,E2 27072.992} C_VEL
LIN {X 0,Y 560.921,Z 1096.009,A -85,B 0,C 180,E1 27071.07,E2 27071.07} C_VEL
LIN {X 0,Y 561.337,Z 1081.332,A -85,B 0,C 180,E1 27069.24,E2 27069.24} C_VEL
LIN {X 0,Y 561.858,Z 1064.769,A -85,B 0,C 180,E1 27067.457,E2 27067.457} C_VEL
LIN {X 0,Y 562.417,Z 1047.631,A -85,B 0,C 180,E1 27065.866,E2 27065.866} C_VEL
LIN {X 0,Y 563.052,Z 1028.915,A -85,B 0,C 180,E1 27064.385,E2 27064.385} C_VEL
LIN {X 0,Y 563.665,Z 1009.913,A -85,B 0,C 180,E1 27063.107,E2 27063.107} C_VEL
LIN {X 0,Y 564.283,Z 989.125,A -85,B 0,C 180,E1 27061.935,E2 27061.935} C_VEL
LIN {X 0,Y 564.891,Z 968.637,A -85,B 0,C 180,E1 27060.99,E2 27060.99} C_VEL
LIN {X 0,Y 565.351,Z 947.31,A -85,B 0,C 180,E1 27060.216,E2 27060.216} C_VEL
LIN {X 0,Y 565.791,Z 925.129,A -85,B 0,C 180,E1 27059.616,E2 27059.616} C_VEL
LIN {X 0,Y 566.063,Z 903.474,A -85,B 0,C 180,E1 27059.216,E2 27059.216} C_VEL
LIN {X 0,Y 567.392,Z 679.442,A -85,B 0,C 180,E1 27056.009,E2 27056.009} C_VEL
LIN {X 0,Y 567.241,Z 677.585,A -85,B 0,C 180,E1 27055.971,E2 27055.971} C_VEL
LIN {X 0,Y 560.514,Z 666.104,A -85,B 0,C 180,E1 27055.318,E2 27055.318} C_VEL
LIN {X 0,Y 560.275,Z 665.01,A -85,B 0,C 180,E1 27055.149,E2 27055.149} C_VEL
LIN {X 0,Y 560.277,Z 664.934,A -85,B 0,C 180,E1 27051.87,E2 27051.87} C_VEL
LIN {X 0,Y 560.262,Z 664.942,A -85,B 0,C 180,E1 27048.542,E2 27048.542} C_VEL
LIN {X 0,Y 560.27,Z 664.945,A -85,B 0,C 180,E1 27045.257,E2 27045.257} C_VEL
LIN {X 0,Y 560.261,Z 664.927,A -85,B 0,C 180,E1 27042.008,E2 27042.008} C_VEL
LIN {X 0,Y 560.263,Z 664.939,A -85,B 0,C 180,E1 27038.753,E2 27038.753} C_VEL
LIN {X 0,Y 560.264,Z 664.935,A -85,B 0,C 180,E1 27035.451,E2 27035.451} C_VEL
LIN {X 0,Y 560.266,Z 664.936,A -85,B 0,C 180,E1 27032.128,E2 27032.128} C_VEL
LIN {X 0,Y 560.277,Z 664.932,A -85,B 0,C 180,E1 27028.806,E2 27028.806} C_VEL
LIN {X 0,Y 560.278,Z 664.938,A -85,B 0,C 180,E1 27025.36,E2 27025.36} C_VEL
LIN {X 0,Y 560.273,Z 664.941,A -85,B 0,C 180,E1 27021.9,E2 27021.9} C_VEL
LIN {X 0,Y 560.278,Z 664.94,A -85,B 0,C 180,E1 27018.629,E2 27018.629} C_VEL
LIN {X 0,Y 560.266,Z 664.94,A -85,B 0,C 180,E1 27015.315,E2 27015.315} C_VEL
LIN {X 0,Y 560.279,Z 664.945,A -85,B 0,C 180,E1 27011.947,E2 27011.947} C_VEL
LIN {X 0,Y 560.262,Z 664.94,A -85,B 0,C 180,E1 27008.622,E2 27008.622} C_VEL
LIN {X 0,Y 560.274,Z 664.947,A -85,B 0,C 180,E1 27005.325,E2 27005.325} C_VEL
LIN {X 0,Y 560.263,Z 664.935,A -85,B 0,C 180,E1 27002.046,E2 27002.046} C_VEL
LIN {X 0,Y 560.267,Z 664.943,A -85,B 0,C 180,E1 26998.773,E2 26998.773} C_VEL
LIN {X 0,Y 560.265,Z 664.94,A -85,B 0,C 180,E1 26995.497,E2 26995.497} C_VEL
LIN {X 0,Y 560.267,Z 664.941,A -85,B 0,C 180,E1 26992.205,E2 26992.205} C_VEL
LIN {X 0,Y 560.272,Z 664.942,A -85,B 0,C 180,E1 26988.888,E2 26988.888} C_VEL
LIN {X 0,Y 560.278,Z 664.936,A -85,B 0,C 180,E1 26985.427,E2 26985.427} C_VEL
LIN {X 0,Y 560.274,Z 664.939,A -85,B 0,C 180,E1 26982.017,E2 26982.017} C_VEL
LIN {X 0,Y 560.266,Z 664.94,A -85,B 0,C 180,E1 26978.65,E2 26978.65} C_VEL
LIN {X 0,Y 560.266,Z 664.939,A -85,B 0,C 180,E1 26975.43,E2 26975.43} C_VEL
LIN {X 0,Y 560.263,Z 664.943,A -85,B 0,C 180,E1 26972.124,E2 26972.124} C_VEL
LIN {X 0,Y 560.262,Z 664.944,A -85,B 0,C 180,E1 26968.833,E2 26968.833} C_VEL
LIN {X 0,Y 560.261,Z 664.937,A -85,B 0,C 180,E1 26965.547,E2 26965.547} C_VEL
LIN {X 0,Y 560.261,Z 664.938,A -85,B 0,C 180,E1 26962.257,E2 26962.257} C_VEL
LIN {X 0,Y 560.261,Z 664.936,A -85,B 0,C 180,E1 26959.014,E2 26959.014} C_VEL
LIN {X 0,Y 560.262,Z 664.935,A -85,B 0,C 180,E1 26955.693,E2 26955.693} C_VEL
LIN {X 0,Y 560.275,Z 664.932,A -85,B 0,C 180,E1 26952.37,E2 26952.37} C_VEL
LIN {X 0,Y 560.327,Z 665.302,A -85,B 0,C 180,E1 26951.863,E2 26951.863} C_VEL
LIN {X 0,Y 563.032,Z 671.58,A -85,B 0,C 180,E1 26951.21,E2 26951.21} C_VEL
LIN {X 0,Y 568.062,Z 682.288,A -85,B 0,C 180,E1 26950.035,E2 26950.035} C_VEL
LIN {X 0,Y 566.908,Z 729.336,A -85,B 0,C 180,E1 26946.97,E2 26946.97} C_VEL
LIN {X 0,Y 566.367,Z 759.679,A -85,B 0,C 180,E1 26945.068,E2 26945.068} C_VEL
LIN {X 0,Y 567.768,Z 769.076,A -85,B 0,C 180,E1 26944.827,E2 26944.827} C_VEL
LIN {X 0,Y 566.349,Z 1004.559,A -85,B 0,C 180,E1 26941.432,E2 26941.432} C_VEL
LIN {X 0,Y 565.94,Z 1066.602,A -85,B 0,C 180,E1 26940.521,E2 26940.521} C_VEL
LIN {X 0,Y 565.548,Z 1088.094,A -85,B 0,C 180,E1 26940.013,E2 26940.013} C_VEL
LIN {X 0,Y 565.084,Z 1109.585,A -85,B 0,C 180,E1 26939.316,E2 26939.316} C_VEL
LIN {X 0,Y 564.575,Z 1130.409,A -85,B 0,C 180,E1 26938.449,E2 26938.449} C_VEL
LIN {X 0,Y 563.938,Z 1150.758,A -85,B 0,C 180,E1 26937.392,E2 26937.392} C_VEL
LIN {X 0,Y 563.302,Z 1171.154,A -85,B 0,C 180,E1 26936.116,E2 26936.116} C_VEL
LIN {X 0,Y 562.699,Z 1189.38,A -85,B 0,C 180,E1 26934.771,E2 26934.771} C_VEL
LIN {X 0,Y 562.101,Z 1207.229,A -85,B 0,C 180,E1 26933.229,E2 26933.229} C_VEL
LIN {X 0,Y 561.575,Z 1223.692,A -85,B 0,C 180,E1 26931.571,E2 26931.571} C_VEL
LIN {X 0,Y 561.083,Z 1239.875,A -85,B 0,C 180,E1 26929.681,E2 26929.681} C_VEL
LIN {X 0,Y 560.709,Z 1254.045,A -85,B 0,C 180,E1 26927.753,E2 26927.753} C_VEL
LIN {X 0,Y 560.406,Z 1266.739,A -85,B 0,C 180,E1 26925.735,E2 26925.735} C_VEL
LIN {X 0,Y 560.197,Z 1277.334,A -85,B 0,C 180,E1 26923.732,E2 26923.732} C_VEL
LIN {X 0,Y 560.057,Z 1287.069,A -85,B 0,C 180,E1 26921.534,E2 26921.534} C_VEL
LIN {X 0,Y 559.979,Z 1294.937,A -85,B 0,C 180,E1 26919.351,E2 26919.351} C_VEL
LIN {X 0,Y 559.928,Z 1300.907,A -85,B 0,C 180,E1 26917.18,E2 26917.18} C_VEL
LIN {X 0,Y 559.906,Z 1305.464,A -85,B 0,C 180,E1 26914.917,E2 26914.917} C_VEL
LIN {X 0,Y 559.899,Z 1308.234,A -85,B 0,C 180,E1 26912.764,E2 26912.764} C_VEL
LIN {X 0,Y 559.894,Z 1309.373,A -85,B 0,C 180,E1 26910.614,E2 26910.614} C_VEL
LIN {X 0,Y 559.895,Z 1309.015,A -85,B 0,C 180,E1 26908.363,E2 26908.363} C_VEL
LIN {X 0,Y 559.899,Z 1307.222,A -85,B 0,C 180,E1 26906.314,E2 26906.314} C_VEL
LIN {X 0,Y 559.909,Z 1303.604,A -85,B 0,C 180,E1 26904.055,E2 26904.055} C_VEL
LIN {X 0,Y 559.945,Z 1298.584,A -85,B 0,C 180,E1 26901.891,E2 26901.891} C_VEL
LIN {X 0,Y 560.004,Z 1292.112,A -85,B 0,C 180,E1 26899.819,E2 26899.819} C_VEL
LIN {X 0,Y 560.107,Z 1283.214,A -85,B 0,C 180,E1 26897.543,E2 26897.543} C_VEL
LIN {X 0,Y 560.282,Z 1273.691,A -85,B 0,C 180,E1 26895.532,E2 26895.532} C_VEL
LIN {X 0,Y 560.515,Z 1262.271,A -85,B 0,C 180,E1 26893.524,E2 26893.524} C_VEL
LIN {X 0,Y 560.841,Z 1248.793,A -85,B 0,C 180,E1 26891.499,E2 26891.499} C_VEL
LIN {X 0,Y 561.233,Z 1234.662,A -85,B 0,C 180,E1 26889.672,E2 26889.672} C_VEL
LIN {X 0,Y 561.727,Z 1218.824,A -85,B 0,C 180,E1 26887.907,E2 26887.907} C_VEL
LIN {X 0,Y 562.275,Z 1202.075,A -85,B 0,C 180,E1 26886.305,E2 26886.305} C_VEL
LIN {X 0,Y 562.893,Z 1183.403,A -85,B 0,C 180,E1 26884.767,E2 26884.767} C_VEL
LIN {X 0,Y 563.512,Z 1164.545,A -85,B 0,C 180,E1 26883.441,E2 26883.441} C_VEL
LIN {X 0,Y 564.136,Z 1144.763,A -85,B 0,C 180,E1 26882.275,E2 26882.275} C_VEL
LIN {X 0,Y 564.713,Z 1124.065,A -85,B 0,C 180,E1 26881.269,E2 26881.269} C_VEL
LIN {X 0,Y 565.261,Z 1102.572,A -85,B 0,C 180,E1 26880.434,E2 26880.434} C_VEL
LIN {X 0,Y 565.682,Z 1081.677,A -85,B 0,C 180,E1 26879.815,E2 26879.815} C_VEL
LIN {X 0,Y 565.984,Z 1060.129,A -85,B 0,C 180,E1 26879.369,E2 26879.369} C_VEL
LIN {X 0,Y 567.35,Z 834.781,A -85,B 0,C 180,E1 26876.131,E2 26876.131} C_VEL
LIN {X 0,Y 567.593,Z 766.671,A -85,B 0,C 180,E1 26875.124,E2 26875.124} C_VEL
LIN {X 0,Y 566.291,Z 759.105,A -85,B 0,C 180,E1 26874.913,E2 26874.913} C_VEL
LIN {X 0,Y 567.427,Z 708.184,A -85,B 0,C 180,E1 26871.667,E2 26871.667} C_VEL
LIN {X 0,Y 568.062,Z 682.288,A -85,B 0,C 180,E1 26869.965,E2 26869.965} C_VEL
LIN {X 0,Y 561.848,Z 668.848,A -85,B 0,C 180,E1 26868.521,E2 26868.521} C_VEL
LIN {X 0,Y 560.326,Z 665.299,A -85,B 0,C 180,E1 26868.137,E2 26868.137} C_VEL
LIN {X 0,Y 560.267,Z 664.931,A -85,B 0,C 180,E1 26867.441,E2 26867.441} C_VEL
LIN {X 0,Y 560.261,Z 664.934,A -85,B 0,C 180,E1 26864.25,E2 26864.25} C_VEL
LIN {X 0,Y 560.261,Z 664.935,A -85,B 0,C 180,E1 26860.986,E2 26860.986} C_VEL
LIN {X 0,Y 560.261,Z 664.938,A -85,B 0,C 180,E1 26857.743,E2 26857.743} C_VEL
LIN {X 0,Y 560.261,Z 664.938,A -85,B 0,C 180,E1 26854.453,E2 26854.453} C_VEL
LIN {X 0,Y 560.262,Z 664.943,A -85,B 0,C 180,E1 26851.261,E2 26851.261} C_VEL
LIN {X 0,Y 560.262,Z 664.944,A -85,B 0,C 180,E1 26847.992,E2 26847.992} C_VEL
LIN {X 0,Y 560.263,Z 664.939,A -85,B 0,C 180,E1 26844.683,E2 26844.683} C_VEL
LIN {X 0,Y 560.263,Z 664.941,A -85,B 0,C 180,E1 26841.46,E2 26841.46} C_VEL
LIN {X 0,Y 560.263,Z 664.936,A -85,B 0,C 180,E1 26838.198,E2 26838.198} C_VEL
LIN {X 0,Y 560.266,Z 664.938,A -85,B 0,C 180,E1 26834.891,E2 26834.891} C_VEL
LIN {X 0,Y 560.275,Z 664.941,A -85,B 0,C 180,E1 26831.529,E2 26831.529} C_VEL
LIN {X 0,Y 560.278,Z 664.936,A -85,B 0,C 180,E1 26828.104,E2 26828.104} C_VEL
LIN {X 0,Y 560.275,Z 664.941,A -85,B 0,C 180,E1 26824.709,E2 26824.709} C_VEL
LIN {X 0,Y 560.272,Z 664.939,A -85,B 0,C 180,E1 26821.431,E2 26821.431} C_VEL
LIN {X 0,Y 560.27,Z 664.936,A -85,B 0,C 180,E1 26818.159,E2 26818.159} C_VEL
LIN {X 0,Y 560.268,Z 664.945,A -85,B 0,C 180,E1 26814.88,E2 26814.88} C_VEL
LIN {X 0,Y 560.266,Z 664.94,A -85,B 0,C 180,E1 26811.585,E2 26811.585} C_VEL
LIN {X 0,Y 560.275,Z 664.943,A -85,B 0,C 180,E1 26808.261,E2 26808.261} C_VEL
LIN {X 0,Y 560.262,Z 664.938,A -85,B 0,C 180,E1 26805.003,E2 26805.003} C_VEL
LIN {X 0,Y 560.28,Z 664.945,A -85,B 0,C 180,E1 26801.688,E2 26801.688} C_VEL
LIN {X 0,Y 560.262,Z 664.939,A -85,B 0,C 180,E1 26798.397,E2 26798.397} C_VEL
LIN {X 0,Y 560.263,Z 664.939,A -85,B 0,C 180,E1 26796.238,E2 26796.238} C_VEL
LIN {X 0,Y 559.283,Z 665.067,A -85,B 0,C 180,E1 26795.45,E2 26795.45} C_VEL
LIN {X 0,Y 552.861,Z 665.869,A -85,B 0,C 180,E1 26793.238,E2 26793.238} C_VEL
LIN {X 0,Y 552.339,Z 665.926,A -85,B 0,C 180,E1 26792.662,E2 26792.662} C_VEL
LIN {X 0,Y 552.343,Z 665.912,A -85,B 0,C 180,E1 26789.297,E2 26789.297} C_VEL
LIN {X 0,Y 552.332,Z 665.929,A -85,B 0,C 180,E1 26785.818,E2 26785.818} C_VEL
LIN {X 0,Y 552.329,Z 665.921,A -85,B 0,C 180,E1 26782.454,E2 26782.454} C_VEL
LIN {X 0,Y 552.328,Z 665.931,A -85,B 0,C 180,E1 26779.171,E2 26779.171} C_VEL
LIN {X 0,Y 552.325,Z 665.933,A -85,B 0,C 180,E1 26775.817,E2 26775.817} C_VEL
LIN {X 0,Y 552.329,Z 665.919,A -85,B 0,C 180,E1 26772.47,E2 26772.47} C_VEL
LIN {X 0,Y 552.325,Z 665.924,A -85,B 0,C 180,E1 26769.18,E2 26769.18} C_VEL
LIN {X 0,Y 552.337,Z 665.904,A -85,B 0,C 180,E1 26765.808,E2 26765.808} C_VEL
LIN {X 0,Y 552.373,Z 666.227,A -85,B 0,C 180,E1 26765.268,E2 26765.268} C_VEL
LIN {X 0,Y 552.864,Z 667.951,A -85,B 0,C 180,E1 26765.101,E2 26765.101} C_VEL
LIN {X 0,Y 560.743,Z 681.251,A -85,B 0,C 180,E1 26764.332,E2 26764.332} C_VEL
LIN {X 0,Y 559.153,Z 905.549,A -85,B 0,C 180,E1 26761.081,E2 26761.081} C_VEL
LIN {X 0,Y 558.848,Z 926.691,A -85,B 0,C 180,E1 26760.675,E2 26760.675} C_VEL
LIN {X 0,Y 558.319,Z 948.661,A -85,B 0,C 180,E1 26760.061,E2 26760.061} C_VEL
LIN {X 0,Y 557.794,Z 969.232,A -85,B 0,C 180,E1 26759.297,E2 26759.297} C_VEL
LIN {X 0,Y 557.091,Z 989.685,A -85,B 0,C 180,E1 26758.34,E2 26758.34} C_VEL
LIN {X 0,Y 556.38,Z 1009.916,A -85,B 0,C 180,E1 26757.183,E2 26757.183} C_VEL
LIN {X 0,Y 555.639,Z 1029.113,A -85,B 0,C 180,E1 26755.876,E2 26755.876} C_VEL
LIN {X 0,Y 554.926,Z 1047.233,A -85,B 0,C 180,E1 26754.425,E2 26754.425} C_VEL
LIN {X 0,Y 554.256,Z 1064.507,A -85,B 0,C 180,E1 26752.805,E2 26752.805} C_VEL
LIN {X 0,Y 553.626,Z 1081.279,A -85,B 0,C 180,E1 26750.979,E2 26750.979} C_VEL
LIN {X 0,Y 553.119,Z 1096.146,A -85,B 0,C 180,E1 26749.098,E2 26749.098} C_VEL
LIN {X 0,Y 552.71,Z 1109.388,A -85,B 0,C 180,E1 26747.149,E2 26747.149} C_VEL
LIN {X 0,Y 552.394,Z 1121.161,A -85,B 0,C 180,E1 26745.108,E2 26745.108} C_VEL
LIN {X 0,Y 552.173,Z 1132.024,A -85,B 0,C 180,E1 26742.869,E2 26742.869} C_VEL
LIN {X 0,Y 552.047,Z 1140.541,A -85,B 0,C 180,E1 26740.751,E2 26740.751} C_VEL
LIN {X 0,Y 551.963,Z 1147.546,A -85,B 0,C 180,E1 26738.542,E2 26738.542} C_VEL
LIN {X 0,Y 551.918,Z 1153.106,A -85,B 0,C 180,E1 26736.24,E2 26736.24} C_VEL
LIN {X 0,Y 551.905,Z 1156.82,A -85,B 0,C 180,E1 26734.051,E2 26734.051} C_VEL
LIN {X 0,Y 551.899,Z 1158.853,A -85,B 0,C 180,E1 26731.869,E2 26731.869} C_VEL
LIN {X 0,Y 551.898,Z 1159.427,A -85,B 0,C 180,E1 26729.585,E2 26729.585} C_VEL
LIN {X 0,Y 551.9,Z 1158.44,A -85,B 0,C 180,E1 26727.404,E2 26727.404} C_VEL
LIN {X 0,Y 551.906,Z 1155.85,A -85,B 0,C 180,E1 26725.22,E2 26725.22} C_VEL
LIN {X 0,Y 551.93,Z 1151.779,A -85,B 0,C 180,E1 26723.029,E2 26723.029} C_VEL
LIN {X 0,Y 551.981,Z 1146.286,A -85,B 0,C 180,E1 26720.933,E2 26720.933} C_VEL
LIN {X 0,Y 552.069,Z 1138.465,A -85,B 0,C 180,E1 26718.615,E2 26718.615} C_VEL
LIN {X 0,Y 552.23,Z 1129.548,A -85,B 0,C 180,E1 26716.479,E2 26716.479} C_VEL
LIN {X 0,Y 552.465,Z 1118.75,A -85,B 0,C 180,E1 26714.356,E2 26714.356} C_VEL
LIN {X 0,Y 552.802,Z 1106.459,A -85,B 0,C 180,E1 26712.311,E2 26712.311} C_VEL
LIN {X 0,Y 553.232,Z 1092.499,A -85,B 0,C 180,E1 26710.323,E2 26710.323} C_VEL
LIN {X 0,Y 553.764,Z 1077.612,A -85,B 0,C 180,E1 26708.499,E2 26708.499} C_VEL
LIN {X 0,Y 554.389,Z 1060.816,A -85,B 0,C 180,E1 26706.736,E2 26706.736} C_VEL
LIN {X 0,Y 555.096,Z 1042.98,A -85,B 0,C 180,E1 26705.128,E2 26705.128} C_VEL
LIN {X 0,Y 555.864,Z 1023.399,A -85,B 0,C 180,E1 26703.623,E2 26703.623} C_VEL
LIN {X 0,Y 556.589,Z 1004.485,A -85,B 0,C 180,E1 26702.39,E2 26702.39} C_VEL
LIN {X 0,Y 557.279,Z 984.789,A -85,B 0,C 180,E1 26701.325,E2 26701.325} C_VEL
LIN {X 0,Y 557.904,Z 964.182,A -85,B 0,C 180,E1 26700.408,E2 26700.408} C_VEL
LIN {X 0,Y 558.524,Z 942.774,A -85,B 0,C 180,E1 26699.661,E2 26699.661} C_VEL
LIN {X 0,Y 558.916,Z 921.036,A -85,B 0,C 180,E1 26699.109,E2 26699.109} C_VEL
LIN {X 0,Y 559.263,Z 892.222,A -85,B 0,C 180,E1 26698.635,E2 26698.635} C_VEL
LIN {X 0,Y 560.706,Z 680.992,A -85,B 0,C 180,E1 26695.571,E2 26695.571} C_VEL
LIN {X 0,Y 553.947,Z 669.808,A -85,B 0,C 180,E1 26694.918,E2 26694.918} C_VEL
LIN {X 0,Y 552.438,Z 666.57,A -85,B 0,C 180,E1 26694.713,E2 26694.713} C_VEL
LIN {X 0,Y 552.335,Z 665.916,A -85,B 0,C 180,E1 26694.474,E2 26694.474} C_VEL
LIN {X 0,Y 552.338,Z 665.92,A -85,B 0,C 180,E1 26691.088,E2 26691.088} C_VEL
LIN {X 0,Y 552.339,Z 665.918,A -85,B 0,C 180,E1 26687.671,E2 26687.671} C_VEL
LIN {X 0,Y 552.326,Z 665.931,A -85,B 0,C 180,E1 26684.328,E2 26684.328} C_VEL
LIN {X 0,Y 552.328,Z 665.934,A -85,B 0,C 180,E1 26680.987,E2 26680.987} C_VEL
LIN {X 0,Y 552.323,Z 665.925,A -85,B 0,C 180,E1 26677.715,E2 26677.715} C_VEL
LIN {X 0,Y 552.325,Z 665.931,A -85,B 0,C 180,E1 26674.389,E2 26674.389} C_VEL
LIN {X 0,Y 552.332,Z 665.92,A -85,B 0,C 180,E1 26671.059,E2 26671.059} C_VEL
LIN {X 0,Y 552.33,Z 665.926,A -85,B 0,C 180,E1 26667.725,E2 26667.725} C_VEL
LIN {X 0,Y 552.344,Z 665.93,A -85,B 0,C 180,E1 26664.263,E2 26664.263} C_VEL
LIN {X 0,Y 552.342,Z 665.927,A -85,B 0,C 180,E1 26660.893,E2 26660.893} C_VEL
LIN {X 0,Y 552.328,Z 665.929,A -85,B 0,C 180,E1 26657.45,E2 26657.45} C_VEL
LIN {X 0,Y 552.34,Z 665.932,A -85,B 0,C 180,E1 26654.145,E2 26654.145} C_VEL
LIN {X 0,Y 552.324,Z 665.926,A -85,B 0,C 180,E1 26650.852,E2 26650.852} C_VEL
LIN {X 0,Y 552.342,Z 665.93,A -85,B 0,C 180,E1 26647.489,E2 26647.489} C_VEL
LIN {X 0,Y 552.327,Z 665.929,A -85,B 0,C 180,E1 26644.114,E2 26644.114} C_VEL
LIN {X 0,Y 552.333,Z 665.932,A -85,B 0,C 180,E1 26640.726,E2 26640.726} C_VEL
LIN {X 0,Y 552.336,Z 665.928,A -85,B 0,C 180,E1 26637.406,E2 26637.406} C_VEL
LIN {X 0,Y 552.337,Z 665.927,A -85,B 0,C 180,E1 26633.973,E2 26633.973} C_VEL
LIN {X 0,Y 552.335,Z 665.938,A -85,B 0,C 180,E1 26630.519,E2 26630.519} C_VEL
LIN {X 0,Y 552.325,Z 665.919,A -85,B 0,C 180,E1 26627.241,E2 26627.241} C_VEL
LIN {X 0,Y 552.325,Z 665.935,A -85,B 0,C 180,E1 26623.921,E2 26623.921} C_VEL
LIN {X 0,Y 552.322,Z 665.919,A -85,B 0,C 180,E1 26620.654,E2 26620.654} C_VEL
LIN {X 0,Y 552.324,Z 665.931,A -85,B 0,C 180,E1 26617.4,E2 26617.4} C_VEL
LIN {X 0,Y 552.323,Z 665.927,A -85,B 0,C 180,E1 26614.116,E2 26614.116} C_VEL
LIN {X 0,Y 552.324,Z 665.921,A -85,B 0,C 180,E1 26610.859,E2 26610.859} C_VEL
LIN {X 0,Y 552.324,Z 665.936,A -85,B 0,C 180,E1 26607.599,E2 26607.599} C_VEL
LIN {X 0,Y 552.323,Z 665.932,A -85,B 0,C 180,E1 26604.345,E2 26604.345} C_VEL
LIN {X 0,Y 552.327,Z 665.933,A -85,B 0,C 180,E1 26601.086,E2 26601.086} C_VEL
LIN {X 0,Y 552.325,Z 665.901,A -85,B 0,C 180,E1 26597.764,E2 26597.764} C_VEL
LIN {X 0,Y 552.347,Z 665.931,A -85,B 0,C 180,E1 26594.324,E2 26594.324} C_VEL
LIN {X 0,Y 552.375,Z 666.203,A -85,B 0,C 180,E1 26592.433,E2 26592.433} C_VEL
LIN {X 0,Y 554.943,Z 672.541,A -85,B 0,C 180,E1 26591.762,E2 26591.762} C_VEL
LIN {X 0,Y 561.473,Z 685.989,A -85,B 0,C 180,E1 26590.344,E2 26590.344} C_VEL
LIN {X 0,Y 560.093,Z 734.033,A -85,B 0,C 180,E1 26587.182,E2 26587.182} C_VEL
LIN {X 0,Y 559.559,Z 759.726,A -85,B 0,C 180,E1 26585.558,E2 26585.558} C_VEL
LIN {X 0,Y 561.19,Z 770.355,A -85,B 0,C 180,E1 26585.276,E2 26585.276} C_VEL
LIN {X 0,Y 559.517,Z 1005.449,A -85,B 0,C 180,E1 26581.847,E2 26581.847} C_VEL
LIN {X 0,Y 559.041,Z 1066.601,A -85,B 0,C 180,E1 26580.939,E2 26580.939} C_VEL
LIN {X 0,Y 558.581,Z 1088.264,A -85,B 0,C 180,E1 26580.422,E2 26580.422} C_VEL
LIN {X 0,Y 558.021,Z 1110.396,A -85,B 0,C 180,E1 26579.691,E2 26579.691} C_VEL
LIN {X 0,Y 557.439,Z 1130.409,A -85,B 0,C 180,E1 26578.848,E2 26578.848} C_VEL
LIN {X 0,Y 556.744,Z 1149.766,A -85,B 0,C 180,E1 26577.835,E2 26577.835} C_VEL
LIN {X 0,Y 555.983,Z 1170.343,A -85,B 0,C 180,E1 26576.544,E2 26576.544} C_VEL
LIN {X 0,Y 555.24,Z 1189.121,A -85,B 0,C 180,E1 26575.149,E2 26575.149} C_VEL
LIN {X 0,Y 554.548,Z 1206.91,A -85,B 0,C 180,E1 26573.594,E2 26573.594} C_VEL
LIN {X 0,Y 553.91,Z 1223.521,A -85,B 0,C 180,E1 26571.903,E2 26571.903} C_VEL
LIN {X 0,Y 553.322,Z 1239.876,A -85,B 0,C 180,E1 26569.969,E2 26569.969} C_VEL
LIN {X 0,Y 552.866,Z 1254.047,A -85,B 0,C 180,E1 26568.014,E2 26568.014} C_VEL
LIN {X 0,Y 552.505,Z 1266.737,A -85,B 0,C 180,E1 26565.966,E2 26565.966} C_VEL
LIN {X 0,Y 552.261,Z 1277.335,A -85,B 0,C 180,E1 26563.933,E2 26563.933} C_VEL
LIN {X 0,Y 552.089,Z 1287.07,A -85,B 0,C 180,E1 26561.703,E2 26561.703} C_VEL
LIN {X 0,Y 551.992,Z 1294.937,A -85,B 0,C 180,E1 26559.487,E2 26559.487} C_VEL
LIN {X 0,Y 551.934,Z 1300.908,A -85,B 0,C 180,E1 26557.285,E2 26557.285} C_VEL
LIN {X 0,Y 551.908,Z 1305.464,A -85,B 0,C 180,E1 26554.989,E2 26554.989} C_VEL
LIN {X 0,Y 551.9,Z 1308.234,A -85,B 0,C 180,E1 26552.804,E2 26552.804} C_VEL
LIN {X 0,Y 551.895,Z 1309.373,A -85,B 0,C 180,E1 26550.623,E2 26550.623} C_VEL
LIN {X 0,Y 551.895,Z 1309.015,A -85,B 0,C 180,E1 26548.339,E2 26548.339} C_VEL
LIN {X 0,Y 551.898,Z 1307.221,A -85,B 0,C 180,E1 26546.261,E2 26546.261} C_VEL
LIN {X 0,Y 551.912,Z 1303.727,A -85,B 0,C 180,E1 26544.031,E2 26544.031} C_VEL
LIN {X 0,Y 551.951,Z 1298.873,A -85,B 0,C 180,E1 26541.877,E2 26541.877} C_VEL
LIN {X 0,Y 552.018,Z 1292.467,A -85,B 0,C 180,E1 26539.776,E2 26539.776} C_VEL
LIN {X 0,Y 552.138,Z 1284.062,A -85,B 0,C 180,E1 26537.556,E2 26537.556} C_VEL
LIN {X 0,Y 552.331,Z 1274.738,A -85,B 0,C 180,E1 26535.534,E2 26535.534} C_VEL
LIN {X 0,Y 552.601,Z 1263.555,A -85,B 0,C 180,E1 26533.497,E2 26533.497} C_VEL
